LIN {X 0,Y 371.368,Z 260.473,A -85,B 0,C 180,E1 -13213.226,E2 -13213.226} C_VEL
LIN {X 0,Y 370.811,Z 274.455,A -85,B 0,C 180,E1 -13213.696,E2 -13213.696} C_VEL
LIN {X 0,Y 369.99,Z 288.054,A -85,B 0,C 180,E1 -13214.366,E2 -13214.366} C_VEL
LIN {X 0,Y 368.934,Z 301.272,A -85,B 0,C 180,E1 -13215.239,E2 -13215.239} C_VEL
LIN {X 0,Y 367.744,Z 313.996,A -85,B 0,C 180,E1 -13216.32,E2 -13216.32} C_VEL
LIN {X 0,Y 366.536,Z 325.561,A -85,B 0,C 180,E1 -13217.543,E2 -13217.543} C_VEL
LIN {X 0,Y 365.255,Z 336.172,A -85,B 0,C 180,E1 -13218.907,E2 -13218.907} C_VEL
LIN {X 0,Y 364.323,Z 345.06,A -85,B 0,C 180,E1 -13220.283,E2 -13220.283} C_VEL
LIN {X 0,Y 363.242,Z 354.016,A -85,B 0,C 180,E1 -13221.937,E2 -13221.937} C_VEL
LIN {X 0,Y 362.182,Z 362.593,A -85,B 0,C 180,E1 -13223.874,E2 -13223.874} C_VEL
LIN {X 0,Y 361.476,Z 368.625,A -85,B 0,C 180,E1 -13225.54,E2 -13225.54} C_VEL
LIN {X 0,Y 360.847,Z 375.044,A -85,B 0,C 180,E1 -13227.768,E2 -13227.768} C_VEL
LIN {X 0,Y 360.557,Z 379.848,A -85,B 0,C 180,E1 -13230,E2 -13230} C_VEL
LIN {X 0,Y 360.321,Z 383.186,A -85,B 0,C 180,E1 -13232.236,E2 -13232.236} C_VEL
LIN {X 0,Y 360.333,Z 385.14,A -85,B 0,C 180,E1 -13234.475,E2 -13234.475} C_VEL
LIN {X 0,Y 360.336,Z 385.758,A -85,B 0,C 180,E1 -13236.721,E2 -13236.721} C_VEL
LIN {X 0,Y 360.251,Z 385.048,A -85,B 0,C 180,E1 -13238.979,E2 -13238.979} C_VEL
LIN {X 0,Y 360.475,Z 382.984,A -85,B 0,C 180,E1 -13241.243,E2 -13241.243} C_VEL
LIN {X 0,Y 360.942,Z 379.51,A -85,B 0,C 180,E1 -13243.513,E2 -13243.513} C_VEL
LIN {X 0,Y 361.492,Z 374.512,A -85,B 0,C 180,E1 -13245.794,E2 -13245.794} C_VEL
LIN {X 0,Y 362.207,Z 369.647,A -85,B 0,C 180,E1 -13247.503,E2 -13247.503} C_VEL
LIN {X 0,Y 363.276,Z 362.599,A -85,B 0,C 180,E1 -13249.495,E2 -13249.495} C_VEL
LIN {X 0,Y 363.491,Z 361.022,A -85,B 0,C 180,E1 -13249.891,E2 -13249.891} C_VEL
LIN {X 0,Y 363.353,Z 357.833,A -85,B 0,C 180,E1 -13250.676,E2 -13250.676} C_VEL
LIN {X 0,Y 361.486,Z 352.461,A -85,B 0,C 180,E1 -13251.961,E2 -13251.961} C_VEL
LIN {X 0,Y 359.701,Z 346.613,A -85,B 0,C 180,E1 -13253.201,E2 -13253.201} C_VEL
LIN {X 0,Y 359.683,Z 342.682,A -85,B 0,C 180,E1 -13253.904,E2 -13253.904} C_VEL
LIN {X 0,Y 361.154,Z 332.979,A -85,B 0,C 180,E1 -13255.348,E2 -13255.348} C_VEL
LIN {X 0,Y 362.74,Z 322.514,A -85,B 0,C 180,E1 -13256.634,E2 -13256.634} C_VEL
LIN {X 0,Y 364.329,Z 309.965,A -85,B 0,C 180,E1 -13257.891,E2 -13257.891} C_VEL
LIN {X 0,Y 365.892,Z 297.682,A -85,B 0,C 180,E1 -13258.855,E2 -13258.855} C_VEL
LIN {X 0,Y 367.075,Z 284.046,A -85,B 0,C 180,E1 -13259.696,E2 -13259.696} C_VEL
LIN {X 0,Y 368.002,Z 270.326,A -85,B 0,C 180,E1 -13260.308,E2 -13260.308} C_VEL
LIN {X 0,Y 368.668,Z 256.311,A -85,B 0,C 180,E1 -13260.71,E2 -13260.71} C_VEL
LIN {X 0,Y 371.022,Z 157.916,A -85,B 0,C 180,E1 -13262.647,E2 -13262.647} C_VEL
LIN {X 0,Y 369.329,Z 151.129,A -85,B 0,C 180,E1 -13262.942,E2 -13262.942} C_VEL
LIN {X 0,Y 360.609,Z 131.607,A -85,B 0,C 180,E1 -13264.169,E2 -13264.169} C_VEL
LIN {X 0,Y 357.38,Z 124.729,A -85,B 0,C 180,E1 -13264.654,E2 -13264.654} C_VEL
LIN {X 0,Y 355.233,Z 116.033,A -85,B 0,C 180,E1 -13267.22,E2 -13267.22} C_VEL
LIN {X 0,Y 354.797,Z 114.414,A -85,B 0,C 180,E1 -13267.739,E2 -13267.739} C_VEL
LIN {X 0,Y 354.768,Z 114.419,A -85,B 0,C 180,E1 -13271.167,E2 -13271.167} C_VEL
LIN {X 0,Y 354.759,Z 114.419,A -85,B 0,C 180,E1 -13274.505,E2 -13274.505} C_VEL
LIN {X 0,Y 354.786,Z 114.42,A -85,B 0,C 180,E1 -13277.661,E2 -13277.661} C_VEL
LIN {X 0,Y 354.786,Z 114.4,A -85,B 0,C 180,E1 -13280.662,E2 -13280.662} C_VEL
LIN {X 0,Y 354.819,Z 114.407,A -85,B 0,C 180,E1 -13284.302,E2 -13284.302} C_VEL
LIN {X 0,Y 354.788,Z 114.416,A -85,B 0,C 180,E1 -13287.666,E2 -13287.666} C_VEL
LIN {X 0,Y 354.801,Z 114.414,A -85,B 0,C 180,E1 -13291.614,E2 -13291.614} C_VEL
LIN {X 0,Y 354.835,Z 114.409,A -85,B 0,C 180,E1 -13295.657,E2 -13295.657} C_VEL
LIN {X 0,Y 354.828,Z 114.412,A -85,B 0,C 180,E1 -13299.113,E2 -13299.113} C_VEL
LIN {X 0,Y 354.881,Z 114.4,A -85,B 0,C 180,E1 -13302.719,E2 -13302.719} C_VEL
LIN {X 0,Y 354.953,Z 114.388,A -85,B 0,C 180,E1 -13306.255,E2 -13306.255} C_VEL
LIN {X 0,Y 354.977,Z 114.392,A -85,B 0,C 180,E1 -13309.736,E2 -13309.736} C_VEL
LIN {X 0,Y 355.103,Z 114.375,A -85,B 0,C 180,E1 -13313.18,E2 -13313.18} C_VEL
LIN {X 0,Y 355.242,Z 114.356,A -85,B 0,C 180,E1 -13317.732,E2 -13317.732} C_VEL
LIN {X 0,Y 355.374,Z 114.338,A -85,B 0,C 180,E1 -13320,E2 -13320} C_VEL
LIN {X 0,Y 355.241,Z 114.355,A -85,B 0,C 180,E1 -13322.267,E2 -13322.267} C_VEL
LIN {X 0,Y 355.09,Z 114.368,A -85,B 0,C 180,E1 -13326.82,E2 -13326.82} C_VEL
LIN {X 0,Y 354.957,Z 114.389,A -85,B 0,C 180,E1 -13330.265,E2 -13330.265} C_VEL
LIN {X 0,Y 354.944,Z 114.395,A -85,B 0,C 180,E1 -13334.019,E2 -13334.019} C_VEL
LIN {X 0,Y 354.923,Z 114.396,A -85,B 0,C 180,E1 -13338.108,E2 -13338.108} C_VEL
LIN {X 0,Y 354.835,Z 114.405,A -85,B 0,C 180,E1 -13342.106,E2 -13342.106} C_VEL
LIN {X 0,Y 354.9,Z 114.397,A -85,B 0,C 180,E1 -13345.827,E2 -13345.827} C_VEL
LIN {X 0,Y 354.854,Z 114.404,A -85,B 0,C 180,E1 -13349.678,E2 -13349.678} C_VEL
LIN {X 0,Y 354.806,Z 114.412,A -85,B 0,C 180,E1 -13353.702,E2 -13353.702} C_VEL
LIN {X 0,Y 354.798,Z 114.413,A -85,B 0,C 180,E1 -13356.459,E2 -13356.459} C_VEL
LIN {X 0,Y 354.824,Z 114.393,A -85,B 0,C 180,E1 -13359.423,E2 -13359.423} C_VEL
LIN {X 0,Y 354.788,Z 114.414,A -85,B 0,C 180,E1 -13362.867,E2 -13362.867} C_VEL
LIN {X 0,Y 354.768,Z 114.417,A -85,B 0,C 180,E1 -13366.104,E2 -13366.104} C_VEL
LIN {X 0,Y 354.789,Z 114.414,A -85,B 0,C 180,E1 -13369.179,E2 -13369.179} C_VEL
LIN {X 0,Y 354.808,Z 114.409,A -85,B 0,C 180,E1 -13372.402,E2 -13372.402} C_VEL
LIN {X 0,Y 354.846,Z 114.473,A -85,B 0,C 180,E1 -13375.237,E2 -13375.237} C_VEL
LIN {X 0,Y 358.014,Z 126.781,A -85,B 0,C 180,E1 -13378.654,E2 -13378.654} C_VEL
LIN {X 0,Y 360.804,Z 138.768,A -85,B 0,C 180,E1 -13381.74,E2 -13381.74} C_VEL
LIN {X 0,Y 364.433,Z 147.556,A -85,B 0,C 180,E1 -13382.271,E2 -13382.271} C_VEL
LIN {X 0,Y 369.54,Z 172.482,A -85,B 0,C 180,E1 -13383.27,E2 -13383.27} C_VEL
LIN {X 0,Y 370.584,Z 178.889,A -85,B 0,C 180,E1 -13383.498,E2 -13383.498} C_VEL
LIN {X 0,Y 368.22,Z 276.377,A -85,B 0,C 180,E1 -13385.435,E2 -13385.435} C_VEL
LIN {X 0,Y 367.273,Z 291.024,A -85,B 0,C 180,E1 -13385.931,E2 -13385.931} C_VEL
LIN {X 0,Y 366.048,Z 304.419,A -85,B 0,C 180,E1 -13386.597,E2 -13386.597} C_VEL
LIN {X 0,Y 364.704,Z 317.241,A -85,B 0,C 180,E1 -13387.458,E2 -13387.458} C_VEL
LIN {X 0,Y 363.113,Z 330.167,A -85,B 0,C 180,E1 -13388.572,E2 -13388.572} C_VEL
LIN {X 0,Y 361.439,Z 341.712,A -85,B 0,C 180,E1 -13389.81,E2 -13389.81} C_VEL
LIN {X 0,Y 359.817,Z 352.311,A -85,B 0,C 180,E1 -13391.199,E2 -13391.199} C_VEL
LIN {X 0,Y 358.132,Z 362.837,A -85,B 0,C 180,E1 -13392.881,E2 -13392.881} C_VEL
LIN {X 0,Y 356.745,Z 371.541,A -85,B 0,C 180,E1 -13394.576,E2 -13394.576} C_VEL
LIN {X 0,Y 355.541,Z 379.91,A -85,B 0,C 180,E1 -13396.569,E2 -13396.569} C_VEL
LIN {X 0,Y 354.459,Z 386.661,A -85,B 0,C 180,E1 -13398.564,E2 -13398.564} C_VEL
LIN {X 0,Y 353.928,Z 391.311,A -85,B 0,C 180,E1 -13400.283,E2 -13400.283} C_VEL
LIN {X 0,Y 353.451,Z 396.148,A -85,B 0,C 180,E1 -13402.574,E2 -13402.574} C_VEL
LIN {X 0,Y 353.281,Z 398.78,A -85,B 0,C 180,E1 -13404.291,E2 -13404.291} C_VEL
LIN {X 0,Y 353.191,Z 401.09,A -85,B 0,C 180,E1 -13406.577,E2 -13406.577} C_VEL
LIN {X 0,Y 353.171,Z 402.06,A -85,B 0,C 180,E1 -13408.86,E2 -13408.86} C_VEL
LIN {X 0,Y 353.188,Z 401.7,A -85,B 0,C 180,E1 -13411.14,E2 -13411.14} C_VEL
LIN {X 0,Y 353.202,Z 399.998,A -85,B 0,C 180,E1 -13413.422,E2 -13413.422} C_VEL
LIN {X 0,Y 353.241,Z 396.911,A -85,B 0,C 180,E1 -13415.709,E2 -13415.709} C_VEL
LIN {X 0,Y 353.48,Z 392.343,A -85,B 0,C 180,E1 -13418,E2 -13418} C_VEL
LIN {X 0,Y 353.8,Z 387.808,A -85,B 0,C 180,E1 -13419.721,E2 -13419.721} C_VEL
LIN {X 0,Y 354.434,Z 381.27,A -85,B 0,C 180,E1 -13421.727,E2 -13421.727} C_VEL
LIN {X 0,Y 355.3,Z 373.143,A -85,B 0,C 180,E1 -13423.731,E2 -13423.731} C_VEL
LIN {X 0,Y 356.161,Z 364.616,A -85,B 0,C 180,E1 -13425.449,E2 -13425.449} C_VEL
LIN {X 0,Y 357.437,Z 354.324,A -85,B 0,C 180,E1 -13427.153,E2 -13427.153} C_VEL
LIN {X 0,Y 358.765,Z 343.962,A -85,B 0,C 180,E1 -13428.562,E2 -13428.562} C_VEL
LIN {X 0,Y 360.083,Z 332.707,A -85,B 0,C 180,E1 -13429.823,E2 -13429.823} C_VEL
LIN {X 0,Y 361.257,Z 320.946,A -85,B 0,C 180,E1 -13430.9,E2 -13430.9} C_VEL
LIN {X 0,Y 362.433,Z 307.882,A -85,B 0,C 180,E1 -13431.843,E2 -13431.843} C_VEL
LIN {X 0,Y 363.526,Z 293.919,A -85,B 0,C 180,E1 -13432.596,E2 -13432.596} C_VEL
LIN {X 0,Y 364.334,Z 279.288,A -85,B 0,C 180,E1 -13433.143,E2 -13433.143} C_VEL
LIN {X 0,Y 364.946,Z 256.943,A -85,B 0,C 180,E1 -13433.628,E2 -13433.628} C_VEL
LIN {X 0,Y 366.399,Z 176.054,A -85,B 0,C 180,E1 -13435.216,E2 -13435.216} C_VEL
LIN {X 0,Y 360.271,Z 140.609,A -85,B 0,C 180,E1 -13436.38,E2 -13436.38} C_VEL
LIN {X 0,Y 359.94,Z 138.758,A -85,B 0,C 180,E1 -13436.465,E2 -13436.465} C_VEL
LIN {X 0,Y 358.697,Z 131.582,A -85,B 0,C 180,E1 -13438.153,E2 -13438.153} C_VEL
LIN {X 0,Y 355.623,Z 117.892,A -85,B 0,C 180,E1 -13441.529,E2 -13441.529} C_VEL
LIN {X 0,Y 354.818,Z 114.415,A -85,B 0,C 180,E1 -13442.456,E2 -13442.456} C_VEL
LIN {X 0,Y 354.821,Z 114.413,A -85,B 0,C 180,E1 -13445.699,E2 -13445.699} C_VEL
LIN {X 0,Y 354.823,Z 114.41,A -85,B 0,C 180,E1 -13449.423,E2 -13449.423} C_VEL
LIN {X 0,Y 354.79,Z 114.413,A -85,B 0,C 180,E1 -13452.868,E2 -13452.868} C_VEL
LIN {X 0,Y 354.851,Z 114.407,A -85,B 0,C 180,E1 -13456.117,E2 -13456.117} C_VEL
LIN {X 0,Y 354.856,Z 114.406,A -85,B 0,C 180,E1 -13459.189,E2 -13459.189} C_VEL
LIN {X 0,Y 354.805,Z 114.41,A -85,B 0,C 180,E1 -13462.403,E2 -13462.403} C_VEL
LIN {X 0,Y 354.81,Z 114.411,A -85,B 0,C 180,E1 -13464.941,E2 -13464.941} C_VEL
LIN {X 0,Y 354.791,Z 114.412,A -85,B 0,C 180,E1 -13468.405,E2 -13468.405} C_VEL
LIN {X 0,Y 354.85,Z 114.408,A -85,B 0,C 180,E1 -13471.619,E2 -13471.619} C_VEL
LIN {X 0,Y 354.898,Z 114.399,A -85,B 0,C 180,E1 -13474.173,E2 -13474.173} C_VEL
LIN {X 0,Y 354.833,Z 114.407,A -85,B 0,C 180,E1 -13477.894,E2 -13477.894} C_VEL
LIN {X 0,Y 354.921,Z 114.395,A -85,B 0,C 180,E1 -13481.892,E2 -13481.892} C_VEL
LIN {X 0,Y 354.941,Z 114.394,A -85,B 0,C 180,E1 -13485.981,E2 -13485.981} C_VEL
LIN {X 0,Y 354.977,Z 114.389,A -85,B 0,C 180,E1 -13489.736,E2 -13489.736} C_VEL
LIN {X 0,Y 355.124,Z 114.371,A -85,B 0,C 180,E1 -13493.181,E2 -13493.181} C_VEL
LIN {X 0,Y 355.243,Z 114.357,A -85,B 0,C 180,E1 -13497.733,E2 -13497.733} C_VEL
LIN {X 0,Y 355.395,Z 114.34,A -85,B 0,C 180,E1 -13500,E2 -13500} C_VEL
LIN {X 0,Y 355.243,Z 114.36,A -85,B 0,C 180,E1 -13502.268,E2 -13502.268} C_VEL
LIN {X 0,Y 355.102,Z 114.374,A -85,B 0,C 180,E1 -13506.82,E2 -13506.82} C_VEL
LIN {X 0,Y 354.977,Z 114.391,A -85,B 0,C 180,E1 -13510.264,E2 -13510.264} C_VEL
LIN {X 0,Y 354.942,Z 114.398,A -85,B 0,C 180,E1 -13514.019,E2 -13514.019} C_VEL
LIN {X 0,Y 354.922,Z 114.397,A -85,B 0,C 180,E1 -13518.109,E2 -13518.109} C_VEL
LIN {X 0,Y 354.835,Z 114.408,A -85,B 0,C 180,E1 -13522.106,E2 -13522.106} C_VEL
LIN {X 0,Y 354.899,Z 114.401,A -85,B 0,C 180,E1 -13525.828,E2 -13525.828} C_VEL
LIN {X 0,Y 354.817,Z 114.411,A -85,B 0,C 180,E1 -13529.682,E2 -13529.682} C_VEL
LIN {X 0,Y 354.806,Z 114.412,A -85,B 0,C 180,E1 -13533.702,E2 -13533.702} C_VEL
LIN {X 0,Y 354.797,Z 114.412,A -85,B 0,C 180,E1 -13536.46,E2 -13536.46} C_VEL
LIN {X 0,Y 354.824,Z 114.411,A -85,B 0,C 180,E1 -13539.424,E2 -13539.424} C_VEL
LIN {X 0,Y 354.789,Z 114.418,A -85,B 0,C 180,E1 -13542.868,E2 -13542.868} C_VEL
LIN {X 0,Y 354.768,Z 114.415,A -85,B 0,C 180,E1 -13546.104,E2 -13546.104} C_VEL
LIN {X 0,Y 354.787,Z 114.414,A -85,B 0,C 180,E1 -13549.179,E2 -13549.179} C_VEL
LIN {X 0,Y 354.807,Z 114.413,A -85,B 0,C 180,E1 -13552.403,E2 -13552.403} C_VEL
LIN {X 0,Y 354.813,Z 114.412,A -85,B 0,C 180,E1 -13554.941,E2 -13554.941} C_VEL
LIN {X 0,Y 354.795,Z 114.418,A -85,B 0,C 180,E1 -13558.406,E2 -13558.406} C_VEL
LIN {X 0,Y 354.803,Z 114.412,A -85,B 0,C 180,E1 -13561.615,E2 -13561.615} C_VEL
LIN {X 0,Y 354.836,Z 114.409,A -85,B 0,C 180,E1 -13565.657,E2 -13565.657} C_VEL
LIN {X 0,Y 354.894,Z 114.59,A -85,B 0,C 180,E1 -13566.745,E2 -13566.745} C_VEL
LIN {X 0,Y 357.071,Z 124.538,A -85,B 0,C 180,E1 -13569.419,E2 -13569.419} C_VEL
LIN {X 0,Y 364.492,Z 143.98,A -85,B 0,C 180,E1 -13570.358,E2 -13570.358} C_VEL
LIN {X 0,Y 366.9,Z 156.799,A -85,B 0,C 180,E1 -13570.79,E2 -13570.79} C_VEL
LIN {X 0,Y 364.744,Z 260.78,A -85,B 0,C 180,E1 -13572.84,E2 -13572.84} C_VEL
LIN {X 0,Y 364.132,Z 275.452,A -85,B 0,C 180,E1 -13573.352,E2 -13573.352} C_VEL
LIN {X 0,Y 363.2,Z 289.405,A -85,B 0,C 180,E1 -13574.066,E2 -13574.066} C_VEL
LIN {X 0,Y 362.109,Z 302.365,A -85,B 0,C 180,E1 -13574.955,E2 -13574.955} C_VEL
LIN {X 0,Y 360.91,Z 314.908,A -85,B 0,C 180,E1 -13576.056,E2 -13576.056} C_VEL
LIN {X 0,Y 359.669,Z 326.341,A -85,B 0,C 180,E1 -13577.301,E2 -13577.301} C_VEL
LIN {X 0,Y 358.271,Z 337.358,A -85,B 0,C 180,E1 -13578.763,E2 -13578.763} C_VEL
LIN {X 0,Y 357.157,Z 347.266,A -85,B 0,C 180,E1 -13580.372,E2 -13580.372} C_VEL
LIN {X 0,Y 356.017,Z 355.883,A -85,B 0,C 180,E1 -13582.057,E2 -13582.057} C_VEL
LIN {X 0,Y 355.031,Z 364.157,A -85,B 0,C 180,E1 -13584.035,E2 -13584.035} C_VEL
LIN {X 0,Y 354.242,Z 370.815,A -85,B 0,C 180,E1 -13586.018,E2 -13586.018} C_VEL
LIN {X 0,Y 353.689,Z 376.731,A -85,B 0,C 180,E1 -13588.292,E2 -13588.292} C_VEL
LIN {X 0,Y 353.47,Z 380.152,A -85,B 0,C 180,E1 -13590,E2 -13590} C_VEL
LIN {X 0,Y 353.224,Z 383.442,A -85,B 0,C 180,E1 -13592.281,E2 -13592.281} C_VEL
LIN {X 0,Y 353.246,Z 385.341,A -85,B 0,C 180,E1 -13594.565,E2 -13594.565} C_VEL
LIN {X 0,Y 353.226,Z 385.912,A -85,B 0,C 180,E1 -13596.856,E2 -13596.856} C_VEL
LIN {X 0,Y 353.163,Z 385.158,A -85,B 0,C 180,E1 -13599.161,E2 -13599.161} C_VEL
LIN {X 0,Y 353.438,Z 383.051,A -85,B 0,C 180,E1 -13601.47,E2 -13601.47} C_VEL
LIN {X 0,Y 353.91,Z 379.531,A -85,B 0,C 180,E1 -13603.786,E2 -13603.786} C_VEL
LIN {X 0,Y 354.52,Z 374.484,A -85,B 0,C 180,E1 -13606.113,E2 -13606.113} C_VEL
LIN {X 0,Y 355.29,Z 369.566,A -85,B 0,C 180,E1 -13607.855,E2 -13607.855} C_VEL
LIN {X 0,Y 356.428,Z 362.461,A -85,B 0,C 180,E1 -13609.885,E2 -13609.885} C_VEL
LIN {X 0,Y 357.633,Z 354.998,A -85,B 0,C 180,E1 -13611.621,E2 -13611.621} C_VEL
LIN {X 0,Y 359.168,Z 345.993,A -85,B 0,C 180,E1 -13613.344,E2 -13613.344} C_VEL
LIN {X 0,Y 359.683,Z 342.682,A -85,B 0,C 180,E1 -13613.904,E2 -13613.904} C_VEL
LIN {X 0,Y 359.684,Z 338.612,A -85,B 0,C 180,E1 -13614.586,E2 -13614.586} C_VEL
LIN {X 0,Y 358.044,Z 331.879,A -85,B 0,C 180,E1 -13615.721,E2 -13615.721} C_VEL
LIN {X 0,Y 356.488,Z 324.785,A -85,B 0,C 180,E1 -13616.791,E2 -13616.791} C_VEL
LIN {X 0,Y 356.6,Z 320.066,A -85,B 0,C 180,E1 -13617.363,E2 -13617.363} C_VEL
LIN {X 0,Y 358.195,Z 307.689,A -85,B 0,C 180,E1 -13618.571,E2 -13618.571} C_VEL
LIN {X 0,Y 359.791,Z 294.774,A -85,B 0,C 180,E1 -13619.553,E2 -13619.553} C_VEL
LIN {X 0,Y 360.938,Z 281.508,A -85,B 0,C 180,E1 -13620.334,E2 -13620.334} C_VEL
LIN {X 0,Y 361.892,Z 267.219,A -85,B 0,C 180,E1 -13620.927,E2 -13620.927} C_VEL
LIN {X 0,Y 362.475,Z 252.016,A -85,B 0,C 180,E1 -13621.315,E2 -13621.315} C_VEL
LIN {X 0,Y 364.784,Z 158.967,A -85,B 0,C 180,E1 -13623.171,E2 -13623.171} C_VEL
LIN {X 0,Y 363.36,Z 153.69,A -85,B 0,C 180,E1 -13623.416,E2 -13623.416} C_VEL
LIN {X 0,Y 355.153,Z 135.268,A -85,B 0,C 180,E1 -13624.608,E2 -13624.608} C_VEL
LIN {X 0,Y 350.218,Z 124.881,A -85,B 0,C 180,E1 -13625.371,E2 -13625.371} C_VEL
LIN {X 0,Y 347.731,Z 115.296,A -85,B 0,C 180,E1 -13628.339,E2 -13628.339} C_VEL
LIN {X 0,Y 347.741,Z 115.295,A -85,B 0,C 180,E1 -13631.832,E2 -13631.832} C_VEL
LIN {X 0,Y 347.701,Z 115.291,A -85,B 0,C 180,E1 -13635.028,E2 -13635.028} C_VEL
LIN {X 0,Y 347.74,Z 115.293,A -85,B 0,C 180,E1 -13638.399,E2 -13638.399} C_VEL
LIN {X 0,Y 347.763,Z 115.291,A -85,B 0,C 180,E1 -13642.014,E2 -13642.014} C_VEL
LIN {X 0,Y 347.744,Z 115.294,A -85,B 0,C 180,E1 -13645.536,E2 -13645.536} C_VEL
LIN {X 0,Y 347.746,Z 115.292,A -85,B 0,C 180,E1 -13648.3,E2 -13648.3} C_VEL
LIN {X 0,Y 347.747,Z 115.29,A -85,B 0,C 180,E1 -13650.984,E2 -13650.984} C_VEL
LIN {X 0,Y 347.749,Z 115.285,A -85,B 0,C 180,E1 -13653.601,E2 -13653.601} C_VEL
LIN {X 0,Y 347.764,Z 115.291,A -85,B 0,C 180,E1 -13656.16,E2 -13656.16} C_VEL
LIN {X 0,Y 347.807,Z 115.285,A -85,B 0,C 180,E1 -13659.909,E2 -13659.909} C_VEL
LIN {X 0,Y 347.833,Z 115.281,A -85,B 0,C 180,E1 -13663.568,E2 -13663.568} C_VEL
LIN {X 0,Y 347.891,Z 115.271,A -85,B 0,C 180,E1 -13667.16,E2 -13667.16} C_VEL
LIN {X 0,Y 347.941,Z 115.258,A -85,B 0,C 180,E1 -13670.701,E2 -13670.701} C_VEL
LIN {X 0,Y 348.053,Z 115.255,A -85,B 0,C 180,E1 -13674.205,E2 -13674.205} C_VEL
LIN {X 0,Y 348.204,Z 115.232,A -85,B 0,C 180,E1 -13677.686,E2 -13677.686} C_VEL
LIN {X 0,Y 348.324,Z 115.216,A -85,B 0,C 180,E1 -13680,E2 -13680} C_VEL
LIN {X 0,Y 348.203,Z 115.232,A -85,B 0,C 180,E1 -13682.313,E2 -13682.313} C_VEL
LIN {X 0,Y 348.056,Z 115.244,A -85,B 0,C 180,E1 -13686.958,E2 -13686.958} C_VEL
LIN {X 0,Y 347.897,Z 115.268,A -85,B 0,C 180,E1 -13690.475,E2 -13690.475} C_VEL
LIN {X 0,Y 347.899,Z 115.272,A -85,B 0,C 180,E1 -13694.15,E2 -13694.15} C_VEL
LIN {X 0,Y 347.891,Z 115.272,A -85,B 0,C 180,E1 -13698.29,E2 -13698.29} C_VEL
LIN {X 0,Y 347.79,Z 115.282,A -85,B 0,C 180,E1 -13701.635,E2 -13701.635} C_VEL
LIN {X 0,Y 347.813,Z 115.276,A -85,B 0,C 180,E1 -13705.108,E2 -13705.108} C_VEL
LIN {X 0,Y 347.811,Z 115.281,A -85,B 0,C 180,E1 -13707.694,E2 -13707.694} C_VEL
LIN {X 0,Y 347.764,Z 115.289,A -85,B 0,C 180,E1 -13710.346,E2 -13710.346} C_VEL
LIN {X 0,Y 347.745,Z 115.295,A -85,B 0,C 180,E1 -13714.464,E2 -13714.464} C_VEL
LIN {X 0,Y 347.773,Z 115.288,A -85,B 0,C 180,E1 -13717.988,E2 -13717.988} C_VEL
LIN {X 0,Y 347.751,Z 115.291,A -85,B 0,C 180,E1 -13721.83,E2 -13721.83} C_VEL
LIN {X 0,Y 347.706,Z 115.286,A -85,B 0,C 180,E1 -13725.027,E2 -13725.027} C_VEL
LIN {X 0,Y 347.751,Z 115.295,A -85,B 0,C 180,E1 -13728.397,E2 -13728.397} C_VEL
LIN {X 0,Y 347.774,Z 115.287,A -85,B 0,C 180,E1 -13732.011,E2 -13732.011} C_VEL
LIN {X 0,Y 347.814,Z 115.462,A -85,B 0,C 180,E1 -13734.662,E2 -13734.662} C_VEL
LIN {X 0,Y 350.854,Z 127.145,A -85,B 0,C 180,E1 -13738.005,E2 -13738.005} C_VEL
LIN {X 0,Y 353.561,Z 138.61,A -85,B 0,C 180,E1 -13741.042,E2 -13741.042} C_VEL
LIN {X 0,Y 358.571,Z 150.353,A -85,B 0,C 180,E1 -13741.794,E2 -13741.794} C_VEL
LIN {X 0,Y 363.378,Z 173.831,A -85,B 0,C 180,E1 -13742.762,E2 -13742.762} C_VEL
LIN {X 0,Y 364.349,Z 179.267,A -85,B 0,C 180,E1 -13742.969,E2 -13742.969} C_VEL
LIN {X 0,Y 361.877,Z 276.592,A -85,B 0,C 180,E1 -13744.937,E2 -13744.937} C_VEL
LIN {X 0,Y 360.891,Z 291.105,A -85,B 0,C 180,E1 -13745.44,E2 -13745.44} C_VEL
LIN {X 0,Y 359.585,Z 304.996,A -85,B 0,C 180,E1 -13746.151,E2 -13746.151} C_VEL
LIN {X 0,Y 358.154,Z 317.742,A -85,B 0,C 180,E1 -13747.029,E2 -13747.029} C_VEL
LIN {X 0,Y 356.525,Z 330.47,A -85,B 0,C 180,E1 -13748.156,E2 -13748.156} C_VEL
LIN {X 0,Y 354.789,Z 341.932,A -85,B 0,C 180,E1 -13749.414,E2 -13749.414} C_VEL
LIN {X 0,Y 353.101,Z 352.464,A -85,B 0,C 180,E1 -13750.828,E2 -13750.828} C_VEL
LIN {X 0,Y 351.319,Z 362.937,A -85,B 0,C 180,E1 -13752.538,E2 -13752.538} C_VEL
LIN {X 0,Y 349.856,Z 371.597,A -85,B 0,C 180,E1 -13754.265,E2 -13754.265} C_VEL
LIN {X 0,Y 348.585,Z 379.925,A -85,B 0,C 180,E1 -13756.296,E2 -13756.296} C_VEL
LIN {X 0,Y 347.468,Z 386.637,A -85,B 0,C 180,E1 -13758.331,E2 -13758.331} C_VEL
LIN {X 0,Y 346.736,Z 392.612,A -85,B 0,C 180,E1 -13760.668,E2 -13760.668} C_VEL
LIN {X 0,Y 346.319,Z 397.016,A -85,B 0,C 180,E1 -13763.006,E2 -13763.006} C_VEL
LIN {X 0,Y 346.138,Z 399.986,A -85,B 0,C 180,E1 -13765.341,E2 -13765.341} C_VEL
LIN {X 0,Y 346.066,Z 401.597,A -85,B 0,C 180,E1 -13767.672,E2 -13767.672} C_VEL
LIN {X 0,Y 346.113,Z 401.878,A -85,B 0,C 180,E1 -13770,E2 -13770} C_VEL
LIN {X 0,Y 346.076,Z 400.823,A -85,B 0,C 180,E1 -13772.328,E2 -13772.328} C_VEL
LIN {X 0,Y 346.128,Z 398.412,A -85,B 0,C 180,E1 -13774.658,E2 -13774.658} C_VEL
LIN {X 0,Y 346.261,Z 394.572,A -85,B 0,C 180,E1 -13776.995,E2 -13776.995} C_VEL
LIN {X 0,Y 346.513,Z 390.635,A -85,B 0,C 180,E1 -13778.749,E2 -13778.749} C_VEL
LIN {X 0,Y 347.073,Z 383.955,A -85,B 0,C 180,E1 -13781.091,E2 -13781.091} C_VEL
LIN {X 0,Y 347.88,Z 376.504,A -85,B 0,C 180,E1 -13783.137,E2 -13783.137} C_VEL
LIN {X 0,Y 348.707,Z 368.798,A -85,B 0,C 180,E1 -13784.866,E2 -13784.866} C_VEL
LIN {X 0,Y 349.944,Z 359.292,A -85,B 0,C 180,E1 -13786.63,E2 -13786.63} C_VEL
LIN {X 0,Y 351.138,Z 348.863,A -85,B 0,C 180,E1 -13788.224,E2 -13788.224} C_VEL
LIN {X 0,Y 352.534,Z 338.664,A -85,B 0,C 180,E1 -13789.507,E2 -13789.507} C_VEL
LIN {X 0,Y 353.955,Z 326.221,A -85,B 0,C 180,E1 -13790.788,E2 -13790.788} C_VEL
LIN {X 0,Y 355.228,Z 314.085,A -85,B 0,C 180,E1 -13791.786,E2 -13791.786} C_VEL
LIN {X 0,Y 356.298,Z 301.099,A -85,B 0,C 180,E1 -13792.621,E2 -13792.621} C_VEL
LIN {X 0,Y 357.289,Z 286.955,A -85,B 0,C 180,E1 -13793.281,E2 -13793.281} C_VEL
LIN {X 0,Y 357.991,Z 272.032,A -85,B 0,C 180,E1 -13793.731,E2 -13793.731} C_VEL
LIN {X 0,Y 359.918,Z 177.39,A -85,B 0,C 180,E1 -13795.62,E2 -13795.62} C_VEL
LIN {X 0,Y 354.009,Z 142.834,A -85,B 0,C 180,E1 -13796.781,E2 -13796.781} C_VEL
LIN {X 0,Y 352.889,Z 138.564,A -85,B 0,C 180,E1 -13796.984,E2 -13796.984} C_VEL
LIN {X 0,Y 350.207,Z 125.859,A -85,B 0,C 180,E1 -13800.112,E2 -13800.112} C_VEL
LIN {X 0,Y 347.779,Z 115.29,A -85,B 0,C 180,E1 -13802.855,E2 -13802.855} C_VEL
LIN {X 0,Y 347.77,Z 115.294,A -85,B 0,C 180,E1 -13806.065,E2 -13806.065} C_VEL
LIN {X 0,Y 347.751,Z 115.291,A -85,B 0,C 180,E1 -13808.792,E2 -13808.792} C_VEL
LIN {X 0,Y 347.75,Z 115.295,A -85,B 0,C 180,E1 -13811.83,E2 -13811.83} C_VEL
LIN {X 0,Y 347.796,Z 115.284,A -85,B 0,C 180,E1 -13815.011,E2 -13815.011} C_VEL
LIN {X 0,Y 347.785,Z 115.286,A -85,B 0,C 180,E1 -13818.39,E2 -13818.39} C_VEL
LIN {X 0,Y 347.772,Z 115.287,A -85,B 0,C 180,E1 -13822.011,E2 -13822.011} C_VEL
LIN {X 0,Y 347.743,Z 115.295,A -85,B 0,C 180,E1 -13825.536,E2 -13825.536} C_VEL
LIN {X 0,Y 347.762,Z 115.29,A -85,B 0,C 180,E1 -13829.654,E2 -13829.654} C_VEL
LIN {X 0,Y 347.85,Z 115.279,A -85,B 0,C 180,E1 -13832.745,E2 -13832.745} C_VEL
LIN {X 0,Y 347.787,Z 115.284,A -85,B 0,C 180,E1 -13836.162,E2 -13836.162} C_VEL
LIN {X 0,Y 347.811,Z 115.282,A -85,B 0,C 180,E1 -13839.909,E2 -13839.909} C_VEL
LIN {X 0,Y 347.865,Z 115.275,A -85,B 0,C 180,E1 -13842.359,E2 -13842.359} C_VEL
LIN {X 0,Y 347.896,Z 115.271,A -85,B 0,C 180,E1 -13845.971,E2 -13845.971} C_VEL
LIN {X 0,Y 347.927,Z 115.267,A -85,B 0,C 180,E1 -13849.526,E2 -13849.526} C_VEL
LIN {X 0,Y 348.09,Z 115.247,A -85,B 0,C 180,E1 -13853.042,E2 -13853.042} C_VEL
LIN {X 0,Y 348.205,Z 115.234,A -85,B 0,C 180,E1 -13857.687,E2 -13857.687} C_VEL
LIN {X 0,Y 348.344,Z 115.218,A -85,B 0,C 180,E1 -13860,E2 -13860} C_VEL
LIN {X 0,Y 348.205,Z 115.236,A -85,B 0,C 180,E1 -13862.314,E2 -13862.314} C_VEL
LIN {X 0,Y 348.069,Z 115.25,A -85,B 0,C 180,E1 -13866.959,E2 -13866.959} C_VEL
LIN {X 0,Y 347.928,Z 115.267,A -85,B 0,C 180,E1 -13870.475,E2 -13870.475} C_VEL
LIN {X 0,Y 347.898,Z 115.274,A -85,B 0,C 180,E1 -13874.15,E2 -13874.15} C_VEL
LIN {X 0,Y 347.89,Z 115.272,A -85,B 0,C 180,E1 -13878.29,E2 -13878.29} C_VEL
LIN {X 0,Y 347.79,Z 115.29,A -85,B 0,C 180,E1 -13881.636,E2 -13881.636} C_VEL
LIN {X 0,Y 347.812,Z 115.283,A -85,B 0,C 180,E1 -13885.109,E2 -13885.109} C_VEL
LIN {X 0,Y 347.808,Z 115.286,A -85,B 0,C 180,E1 -13887.694,E2 -13887.694} C_VEL
LIN {X 0,Y 347.749,Z 115.289,A -85,B 0,C 180,E1 -13890.348,E2 -13890.348} C_VEL
LIN {X 0,Y 347.748,Z 115.29,A -85,B 0,C 180,E1 -13894.044,E2 -13894.044} C_VEL
LIN {X 0,Y 347.761,Z 115.291,A -85,B 0,C 180,E1 -13897.321,E2 -13897.321} C_VEL
LIN {X 0,Y 347.732,Z 115.293,A -85,B 0,C 180,E1 -13900.297,E2 -13900.297} C_VEL
LIN {X 0,Y 347.727,Z 115.294,A -85,B 0,C 180,E1 -13903.408,E2 -13903.408} C_VEL
LIN {X 0,Y 347.726,Z 115.297,A -85,B 0,C 180,E1 -13906.687,E2 -13906.687} C_VEL
LIN {X 0,Y 347.747,Z 115.291,A -85,B 0,C 180,E1 -13910.174,E2 -13910.174} C_VEL
LIN {X 0,Y 347.761,Z 115.293,A -85,B 0,C 180,E1 -13912.68,E2 -13912.68} C_VEL
LIN {X 0,Y 347.749,Z 115.291,A -85,B 0,C 180,E1 -13915.957,E2 -13915.957} C_VEL
LIN {X 0,Y 347.742,Z 115.292,A -85,B 0,C 180,E1 -13919.652,E2 -13919.652} C_VEL
LIN {X 0,Y 347.752,Z 115.29,A -85,B 0,C 180,E1 -13923.602,E2 -13923.602} C_VEL
LIN {X 0,Y 347.843,Z 115.401,A -85,B 0,C 180,E1 -13926.324,E2 -13926.324} C_VEL
LIN {X 0,Y 349.958,Z 124.852,A -85,B 0,C 180,E1 -13928.896,E2 -13928.896} C_VEL
LIN {X 0,Y 357.973,Z 145.511,A -85,B 0,C 180,E1 -13929.936,E2 -13929.936} C_VEL
LIN {X 0,Y 360.385,Z 157.192,A -85,B 0,C 180,E1 -13930.356,E2 -13930.356} C_VEL
LIN {X 0,Y 358.115,Z 261.076,A -85,B 0,C 180,E1 -13932.438,E2 -13932.438} C_VEL
LIN {X 0,Y 357.504,Z 275.688,A -85,B 0,C 180,E1 -13932.96,E2 -13932.96} C_VEL
LIN {X 0,Y 356.536,Z 289.624,A -85,B 0,C 180,E1 -13933.687,E2 -13933.687} C_VEL
LIN {X 0,Y 355.306,Z 303.452,A -85,B 0,C 180,E1 -13934.659,E2 -13934.659} C_VEL
LIN {X 0,Y 354.087,Z 315.814,A -85,B 0,C 180,E1 -13935.782,E2 -13935.782} C_VEL
LIN {X 0,Y 352.656,Z 328.28,A -85,B 0,C 180,E1 -13937.191,E2 -13937.191} C_VEL
LIN {X 0,Y 351.352,Z 338.184,A -85,B 0,C 180,E1 -13938.562,E2 -13938.562} C_VEL
LIN {X 0,Y 350.193,Z 347.856,A -85,B 0,C 180,E1 -13940.178,E2 -13940.178} C_VEL
LIN {X 0,Y 349.01,Z 356.403,A -85,B 0,C 180,E1 -13941.897,E2 -13941.897} C_VEL
LIN {X 0,Y 348.013,Z 364.601,A -85,B 0,C 180,E1 -13943.914,E2 -13943.914} C_VEL
LIN {X 0,Y 347.19,Z 371.198,A -85,B 0,C 180,E1 -13945.937,E2 -13945.937} C_VEL
LIN {X 0,Y 346.617,Z 377.058,A -85,B 0,C 180,E1 -13948.257,E2 -13948.257} C_VEL
LIN {X 0,Y 346.385,Z 380.456,A -85,B 0,C 180,E1 -13950,E2 -13950} C_VEL
LIN {X 0,Y 346.131,Z 383.688,A -85,B 0,C 180,E1 -13952.328,E2 -13952.328} C_VEL
LIN {X 0,Y 346.144,Z 385.536,A -85,B 0,C 180,E1 -13954.659,E2 -13954.659} C_VEL
LIN {X 0,Y 346.199,Z 385.972,A -85,B 0,C 180,E1 -13955.885,E2 -13955.885} C_VEL
LIN {X 0,Y 346.087,Z 385.834,A -85,B 0,C 180,E1 -13958.172,E2 -13958.172} C_VEL
LIN {X 0,Y 346.163,Z 384.365,A -85,B 0,C 180,E1 -13960.529,E2 -13960.529} C_VEL
LIN {X 0,Y 346.642,Z 381.518,A -85,B 0,C 180,E1 -13962.887,E2 -13962.887} C_VEL
LIN {X 0,Y 347.172,Z 377.206,A -85,B 0,C 180,E1 -13965.258,E2 -13965.258} C_VEL
LIN {X 0,Y 348.123,Z 371.286,A -85,B 0,C 180,E1 -13967.627,E2 -13967.627} C_VEL
LIN {X 0,Y 349.249,Z 364.573,A -85,B 0,C 180,E1 -13969.698,E2 -13969.698} C_VEL
LIN {X 0,Y 350.663,Z 356.166,A -85,B 0,C 180,E1 -13971.764,E2 -13971.764} C_VEL
LIN {X 0,Y 352.234,Z 347.367,A -85,B 0,C 180,E1 -13973.519,E2 -13973.519} C_VEL
LIN {X 0,Y 353.946,Z 336.656,A -85,B 0,C 180,E1 -13975.272,E2 -13975.272} C_VEL
LIN {X 0,Y 355.694,Z 325.806,A -85,B 0,C 180,E1 -13976.712,E2 -13976.712} C_VEL
LIN {X 0,Y 356.6,Z 320.066,A -85,B 0,C 180,E1 -13977.363,E2 -13977.363} C_VEL
LIN {X 0,Y 356.443,Z 316.886,A -85,B 0,C 180,E1 -13977.75,E2 -13977.75} C_VEL
LIN {X 0,Y 352.515,Z 306.935,A -85,B 0,C 180,E1 -13979.092,E2 -13979.092} C_VEL
LIN {X 0,Y 352.36,Z 303.512,A -85,B 0,C 180,E1 -13979.419,E2 -13979.419} C_VEL
LIN {X 0,Y 353.796,Z 290.433,A -85,B 0,C 180,E1 -13980.352,E2 -13980.352} C_VEL
LIN {X 0,Y 354.997,Z 276.305,A -85,B 0,C 180,E1 -13981.102,E2 -13981.102} C_VEL
LIN {X 0,Y 355.889,Z 261.563,A -85,B 0,C 180,E1 -13981.63,E2 -13981.63} C_VEL
LIN {X 0,Y 358.698,Z 160.682,A -85,B 0,C 180,E1 -13983.687,E2 -13983.687} C_VEL
LIN {X 0,Y 357.493,Z 156.399,A -85,B 0,C 180,E1 -13983.897,E2 -13983.897} C_VEL
LIN {X 0,Y 349.512,Z 138.471,A -85,B 0,C 180,E1 -13985.092,E2 -13985.092} C_VEL
LIN {X 0,Y 343.035,Z 125.173,A -85,B 0,C 180,E1 -13986.09,E2 -13986.09} C_VEL
LIN {X 0,Y 340.694,Z 116.172,A -85,B 0,C 180,E1 -13988.968,E2 -13988.968} C_VEL
LIN {X 0,Y 340.673,Z 116.174,A -85,B 0,C 180,E1 -13992.905,E2 -13992.905} C_VEL
LIN {X 0,Y 340.673,Z 116.171,A -85,B 0,C 180,E1 -13997.095,E2 -13997.095} C_VEL
LIN {X 0,Y 340.656,Z 116.158,A -85,B 0,C 180,E1 -14000.241,E2 -14000.241} C_VEL
LIN {X 0,Y 340.708,Z 116.167,A -85,B 0,C 180,E1 -14003.56,E2 -14003.56} C_VEL
LIN {X 0,Y 340.693,Z 116.17,A -85,B 0,C 180,E1 -14006.153,E2 -14006.153} C_VEL
LIN {X 0,Y 340.725,Z 116.161,A -85,B 0,C 180,E1 -14010.034,E2 -14010.034} C_VEL
LIN {X 0,Y 340.72,Z 116.164,A -85,B 0,C 180,E1 -14013.012,E2 -14013.012} C_VEL
LIN {X 0,Y 340.74,Z 116.165,A -85,B 0,C 180,E1 -14015.637,E2 -14015.637} C_VEL
LIN {X 0,Y 340.735,Z 116.166,A -85,B 0,C 180,E1 -14019.473,E2 -14019.473} C_VEL
LIN {X 0,Y 340.794,Z 116.149,A -85,B 0,C 180,E1 -14021.98,E2 -14021.98} C_VEL
LIN {X 0,Y 340.871,Z 116.144,A -85,B 0,C 180,E1 -14025.705,E2 -14025.705} C_VEL
LIN {X 0,Y 340.871,Z 116.148,A -85,B 0,C 180,E1 -14029.306,E2 -14029.306} C_VEL
LIN {X 0,Y 341.012,Z 116.131,A -85,B 0,C 180,E1 -14032.897,E2 -14032.897} C_VEL
LIN {X 0,Y 340.834,Z 116.149,A -85,B 0,C 180,E1 -14035.269,E2 -14035.269} C_VEL
LIN {X 0,Y 341.165,Z 116.108,A -85,B 0,C 180,E1 -14037.639,E2 -14037.639} C_VEL
LIN {X 0,Y 341.275,Z 116.094,A -85,B 0,C 180,E1 -14040,E2 -14040} C_VEL
LIN {X 0,Y 341.165,Z 116.109,A -85,B 0,C 180,E1 -14042.361,E2 -14042.361} C_VEL
LIN {X 0,Y 341.003,Z 116.123,A -85,B 0,C 180,E1 -14047.103,E2 -14047.103} C_VEL
LIN {X 0,Y 340.849,Z 116.146,A -85,B 0,C 180,E1 -14050.694,E2 -14050.694} C_VEL
LIN {X 0,Y 340.864,Z 116.148,A -85,B 0,C 180,E1 -14054.325,E2 -14054.325} C_VEL
LIN {X 0,Y 340.838,Z 116.151,A -85,B 0,C 180,E1 -14058.466,E2 -14058.466} C_VEL
LIN {X 0,Y 340.754,Z 116.16,A -85,B 0,C 180,E1 -14061.857,E2 -14061.857} C_VEL
LIN {X 0,Y 340.773,Z 116.156,A -85,B 0,C 180,E1 -14065.664,E2 -14065.664} C_VEL
LIN {X 0,Y 340.742,Z 116.16,A -85,B 0,C 180,E1 -14068.319,E2 -14068.319} C_VEL
LIN {X 0,Y 340.704,Z 116.169,A -85,B 0,C 180,E1 -14071.044,E2 -14071.044} C_VEL
LIN {X 0,Y 340.718,Z 116.163,A -85,B 0,C 180,E1 -14075.279,E2 -14075.279} C_VEL
LIN {X 0,Y 340.709,Z 116.16,A -85,B 0,C 180,E1 -14078.386,E2 -14078.386} C_VEL
LIN {X 0,Y 340.699,Z 116.171,A -85,B 0,C 180,E1 -14082.045,E2 -14082.045} C_VEL
LIN {X 0,Y 340.652,Z 116.176,A -85,B 0,C 180,E1 -14086.227,E2 -14086.227} C_VEL
LIN {X 0,Y 340.689,Z 116.171,A -85,B 0,C 180,E1 -14089.753,E2 -14089.753} C_VEL
LIN {X 0,Y 340.706,Z 116.167,A -85,B 0,C 180,E1 -14093.258,E2 -14093.258} C_VEL
LIN {X 0,Y 340.771,Z 116.257,A -85,B 0,C 180,E1 -14094,E2 -14094} C_VEL
LIN {X 0,Y 343.421,Z 126.529,A -85,B 0,C 180,E1 -14097.04,E2 -14097.04} C_VEL
LIN {X 0,Y 346.172,Z 137.811,A -85,B 0,C 180,E1 -14100.189,E2 -14100.189} C_VEL
LIN {X 0,Y 346.393,Z 138.621,A -85,B 0,C 180,E1 -14100.321,E2 -14100.321} C_VEL
LIN {X 0,Y 352.712,Z 152.863,A -85,B 0,C 180,E1 -14101.291,E2 -14101.291} C_VEL
LIN {X 0,Y 357.62,Z 177.455,A -85,B 0,C 180,E1 -14102.322,E2 -14102.322} C_VEL
LIN {X 0,Y 358.162,Z 181.496,A -85,B 0,C 180,E1 -14102.463,E2 -14102.463} C_VEL
LIN {X 0,Y 355.58,Z 276.806,A -85,B 0,C 180,E1 -14104.422,E2 -14104.422} C_VEL
LIN {X 0,Y 354.564,Z 291.192,A -85,B 0,C 180,E1 -14104.932,E2 -14104.932} C_VEL
LIN {X 0,Y 353.141,Z 305.581,A -85,B 0,C 180,E1 -14105.688,E2 -14105.688} C_VEL
LIN {X 0,Y 351.615,Z 318.392,A -85,B 0,C 180,E1 -14106.597,E2 -14106.597} C_VEL
LIN {X 0,Y 349.944,Z 330.777,A -85,B 0,C 180,E1 -14107.724,E2 -14107.724} C_VEL
LIN {X 0,Y 347.953,Z 343.325,A -85,B 0,C 180,E1 -14109.146,E2 -14109.146} C_VEL
LIN {X 0,Y 346.06,Z 354.534,A -85,B 0,C 180,E1 -14110.73,E2 -14110.73} C_VEL
LIN {X 0,Y 344.252,Z 364.583,A -85,B 0,C 180,E1 -14112.475,E2 -14112.475} C_VEL
LIN {X 0,Y 342.762,Z 372.945,A -85,B 0,C 180,E1 -14114.236,E2 -14114.236} C_VEL
LIN {X 0,Y 341.509,Z 380.951,A -85,B 0,C 180,E1 -14116.31,E2 -14116.31} C_VEL
LIN {X 0,Y 340.492,Z 386.609,A -85,B 0,C 180,E1 -14118.088,E2 -14118.088} C_VEL
LIN {X 0,Y 339.7,Z 392.548,A -85,B 0,C 180,E1 -14120.473,E2 -14120.473} C_VEL
LIN {X 0,Y 339.246,Z 396.925,A -85,B 0,C 180,E1 -14122.86,E2 -14122.86} C_VEL
LIN {X 0,Y 339.043,Z 399.868,A -85,B 0,C 180,E1 -14125.244,E2 -14125.244} C_VEL
LIN {X 0,Y 338.981,Z 401.453,A -85,B 0,C 180,E1 -14127.623,E2 -14127.623} C_VEL
LIN {X 0,Y 339.015,Z 401.708,A -85,B 0,C 180,E1 -14130,E2 -14130} C_VEL
LIN {X 0,Y 338.99,Z 400.628,A -85,B 0,C 180,E1 -14132.376,E2 -14132.376} C_VEL
LIN {X 0,Y 339.048,Z 399.583,A -85,B 0,C 180,E1 -14133.565,E2 -14133.565} C_VEL
LIN {X 0,Y 339.087,Z 396.441,A -85,B 0,C 180,E1 -14135.948,E2 -14135.948} C_VEL
LIN {X 0,Y 339.335,Z 391.794,A -85,B 0,C 180,E1 -14138.336,E2 -14138.336} C_VEL
LIN {X 0,Y 339.695,Z 387.219,A -85,B 0,C 180,E1 -14140.128,E2 -14140.128} C_VEL
LIN {X 0,Y 340.421,Z 380.615,A -85,B 0,C 180,E1 -14142.217,E2 -14142.217} C_VEL
LIN {X 0,Y 341.354,Z 372.403,A -85,B 0,C 180,E1 -14144.304,E2 -14144.304} C_VEL
LIN {X 0,Y 342.379,Z 363.793,A -85,B 0,C 180,E1 -14146.088,E2 -14146.088} C_VEL
LIN {X 0,Y 343.776,Z 353.357,A -85,B 0,C 180,E1 -14147.857,E2 -14147.857} C_VEL
LIN {X 0,Y 345.056,Z 344.032,A -85,B 0,C 180,E1 -14149.173,E2 -14149.173} C_VEL
LIN {X 0,Y 346.501,Z 332.868,A -85,B 0,C 180,E1 -14150.48,E2 -14150.48} C_VEL
LIN {X 0,Y 347.831,Z 320.542,A -85,B 0,C 180,E1 -14151.652,E2 -14151.652} C_VEL
LIN {X 0,Y 349.079,Z 307.2,A -85,B 0,C 180,E1 -14152.646,E2 -14152.646} C_VEL
LIN {X 0,Y 350.27,Z 293.115,A -85,B 0,C 180,E1 -14153.423,E2 -14153.423} C_VEL
LIN {X 0,Y 351.16,Z 278.253,A -85,B 0,C 180,E1 -14153.987,E2 -14153.987} C_VEL
LIN {X 0,Y 351.845,Z 253.688,A -85,B 0,C 180,E1 -14154.525,E2 -14154.525} C_VEL
LIN {X 0,Y 353.357,Z 178.213,A -85,B 0,C 180,E1 -14156.057,E2 -14156.057} C_VEL
LIN {X 0,Y 347.704,Z 144.701,A -85,B 0,C 180,E1 -14157.208,E2 -14157.208} C_VEL
LIN {X 0,Y 345.652,Z 138.445,A -85,B 0,C 180,E1 -14157.52,E2 -14157.52} C_VEL
LIN {X 0,Y 342.895,Z 125.407,A -85,B 0,C 180,E1 -14160.824,E2 -14160.824} C_VEL
LIN {X 0,Y 340.71,Z 116.171,A -85,B 0,C 180,E1 -14163.312,E2 -14163.312} C_VEL
LIN {X 0,Y 340.704,Z 116.17,A -85,B 0,C 180,E1 -14166.741,E2 -14166.741} C_VEL
LIN {X 0,Y 340.687,Z 116.173,A -85,B 0,C 180,E1 -14170.247,E2 -14170.247} C_VEL
LIN {X 0,Y 340.676,Z 116.177,A -85,B 0,C 180,E1 -14173.777,E2 -14173.777} C_VEL
LIN {X 0,Y 340.74,Z 116.163,A -85,B 0,C 180,E1 -14177.106,E2 -14177.106} C_VEL
LIN {X 0,Y 340.732,Z 116.162,A -85,B 0,C 180,E1 -14180.252,E2 -14180.252} C_VEL
LIN {X 0,Y 340.709,Z 116.171,A -85,B 0,C 180,E1 -14183.559,E2 -14183.559} C_VEL
LIN {X 0,Y 340.691,Z 116.168,A -85,B 0,C 180,E1 -14186.153,E2 -14186.153} C_VEL
LIN {X 0,Y 340.773,Z 116.158,A -85,B 0,C 180,E1 -14190.332,E2 -14190.332} C_VEL
LIN {X 0,Y 340.803,Z 116.159,A -85,B 0,C 180,E1 -14193.02,E2 -14193.02} C_VEL
LIN {X 0,Y 340.727,Z 116.167,A -85,B 0,C 180,E1 -14196.927,E2 -14196.927} C_VEL
LIN {X 0,Y 340.789,Z 116.16,A -85,B 0,C 180,E1 -14200.734,E2 -14200.734} C_VEL
LIN {X 0,Y 340.786,Z 116.16,A -85,B 0,C 180,E1 -14203.219,E2 -14203.219} C_VEL
LIN {X 0,Y 340.843,Z 116.152,A -85,B 0,C 180,E1 -14206.891,E2 -14206.891} C_VEL
LIN {X 0,Y 340.923,Z 116.145,A -85,B 0,C 180,E1 -14210.508,E2 -14210.508} C_VEL
LIN {X 0,Y 341.058,Z 116.124,A -85,B 0,C 180,E1 -14212.898,E2 -14212.898} C_VEL
LIN {X 0,Y 341.167,Z 116.11,A -85,B 0,C 180,E1 -14217.639,E2 -14217.639} C_VEL
LIN {X 0,Y 341.294,Z 116.096,A -85,B 0,C 180,E1 -14220,E2 -14220} C_VEL
LIN {X 0,Y 341.167,Z 116.112,A -85,B 0,C 180,E1 -14222.361,E2 -14222.361} C_VEL
LIN {X 0,Y 341.017,Z 116.128,A -85,B 0,C 180,E1 -14227.103,E2 -14227.103} C_VEL
LIN {X 0,Y 340.87,Z 116.145,A -85,B 0,C 180,E1 -14230.694,E2 -14230.694} C_VEL
LIN {X 0,Y 340.862,Z 116.149,A -85,B 0,C 180,E1 -14234.325,E2 -14234.325} C_VEL
LIN {X 0,Y 340.836,Z 116.149,A -85,B 0,C 180,E1 -14238.467,E2 -14238.467} C_VEL
LIN {X 0,Y 340.753,Z 116.164,A -85,B 0,C 180,E1 -14241.857,E2 -14241.857} C_VEL
LIN {X 0,Y 340.772,Z 116.162,A -85,B 0,C 180,E1 -14245.665,E2 -14245.665} C_VEL
LIN {X 0,Y 340.728,Z 116.165,A -85,B 0,C 180,E1 -14248.321,E2 -14248.321} C_VEL
LIN {X 0,Y 340.697,Z 116.171,A -85,B 0,C 180,E1 -14251.045,E2 -14251.045} C_VEL
LIN {X 0,Y 340.718,Z 116.169,A -85,B 0,C 180,E1 -14255.279,E2 -14255.279} C_VEL
LIN {X 0,Y 340.709,Z 116.167,A -85,B 0,C 180,E1 -14258.386,E2 -14258.386} C_VEL
LIN {X 0,Y 340.699,Z 116.167,A -85,B 0,C 180,E1 -14262.046,E2 -14262.046} C_VEL
LIN {X 0,Y 340.682,Z 116.17,A -85,B 0,C 180,E1 -14265.462,E2 -14265.462} C_VEL
LIN {X 0,Y 340.686,Z 116.174,A -85,B 0,C 180,E1 -14268.691,E2 -14268.691} C_VEL
LIN {X 0,Y 340.733,Z 116.161,A -85,B 0,C 180,E1 -14271.773,E2 -14271.773} C_VEL
LIN {X 0,Y 340.724,Z 116.165,A -85,B 0,C 180,E1 -14275.596,E2 -14275.596} C_VEL
LIN {X 0,Y 340.696,Z 116.17,A -85,B 0,C 180,E1 -14278.955,E2 -14278.955} C_VEL
LIN {X 0,Y 340.722,Z 116.165,A -85,B 0,C 180,E1 -14283.013,E2 -14283.013} C_VEL
LIN {X 0,Y 340.769,Z 116.214,A -85,B 0,C 180,E1 -14285.883,E2 -14285.883} C_VEL
LIN {X 0,Y 342.775,Z 125.107,A -85,B 0,C 180,E1 -14288.343,E2 -14288.343} C_VEL
LIN {X 0,Y 350.721,Z 145.003,A -85,B 0,C 180,E1 -14289.399,E2 -14289.399} C_VEL
LIN {X 0,Y 352.438,Z 150.772,A -85,B 0,C 180,E1 -14289.652,E2 -14289.652} C_VEL
LIN {X 0,Y 353.858,Z 158.628,A -85,B 0,C 180,E1 -14289.927,E2 -14289.927} C_VEL
LIN {X 0,Y 351.514,Z 261.347,A -85,B 0,C 180,E1 -14292.022,E2 -14292.022} C_VEL
LIN {X 0,Y 350.893,Z 275.912,A -85,B 0,C 180,E1 -14292.554,E2 -14292.554} C_VEL
LIN {X 0,Y 349.897,Z 289.831,A -85,B 0,C 180,E1 -14293.293,E2 -14293.293} C_VEL
LIN {X 0,Y 348.727,Z 302.77,A -85,B 0,C 180,E1 -14294.213,E2 -14294.213} C_VEL
LIN {X 0,Y 347.43,Z 315.299,A -85,B 0,C 180,E1 -14295.354,E2 -14295.354} C_VEL
LIN {X 0,Y 346.056,Z 326.726,A -85,B 0,C 180,E1 -14296.644,E2 -14296.644} C_VEL
LIN {X 0,Y 344.497,Z 338.193,A -85,B 0,C 180,E1 -14298.229,E2 -14298.229} C_VEL
LIN {X 0,Y 343.237,Z 348.44,A -85,B 0,C 180,E1 -14299.977,E2 -14299.977} C_VEL
LIN {X 0,Y 342.008,Z 356.919,A -85,B 0,C 180,E1 -14301.73,E2 -14301.73} C_VEL
LIN {X 0,Y 340.98,Z 365.031,A -85,B 0,C 180,E1 -14303.788,E2 -14303.788} C_VEL
LIN {X 0,Y 340.14,Z 371.571,A -85,B 0,C 180,E1 -14305.853,E2 -14305.853} C_VEL
LIN {X 0,Y 339.549,Z 377.383,A -85,B 0,C 180,E1 -14308.221,E2 -14308.221} C_VEL
LIN {X 0,Y 339.285,Z 380.752,A -85,B 0,C 180,E1 -14310,E2 -14310} C_VEL
LIN {X 0,Y 339.042,Z 383.926,A -85,B 0,C 180,E1 -14312.376,E2 -14312.376} C_VEL
LIN {X 0,Y 339.047,Z 385.731,A -85,B 0,C 180,E1 -14314.756,E2 -14314.756} C_VEL
LIN {X 0,Y 339.095,Z 386.138,A -85,B 0,C 180,E1 -14315.948,E2 -14315.948} C_VEL
LIN {X 0,Y 338.989,Z 385.966,A -85,B 0,C 180,E1 -14318.345,E2 -14318.345} C_VEL
LIN {X 0,Y 339.113,Z 384.455,A -85,B 0,C 180,E1 -14320.75,E2 -14320.75} C_VEL
LIN {X 0,Y 339.626,Z 381.563,A -85,B 0,C 180,E1 -14323.158,E2 -14323.158} C_VEL
LIN {X 0,Y 340.206,Z 377.206,A -85,B 0,C 180,E1 -14325.578,E2 -14325.578} C_VEL
LIN {X 0,Y 340.937,Z 372.859,A -85,B 0,C 180,E1 -14327.392,E2 -14327.392} C_VEL
LIN {X 0,Y 342.057,Z 366.51,A -85,B 0,C 180,E1 -14329.504,E2 -14329.504} C_VEL
LIN {X 0,Y 343.454,Z 358.574,A -85,B 0,C 180,E1 -14331.613,E2 -14331.613} C_VEL
LIN {X 0,Y 345.062,Z 350.092,A -85,B 0,C 180,E1 -14333.434,E2 -14333.434} C_VEL
LIN {X 0,Y 346.765,Z 340.169,A -85,B 0,C 180,E1 -14335.19,E2 -14335.19} C_VEL
LIN {X 0,Y 348.667,Z 328.907,A -85,B 0,C 180,E1 -14336.809,E2 -14336.809} C_VEL
LIN {X 0,Y 350.618,Z 316.625,A -85,B 0,C 180,E1 -14338.218,E2 -14338.218} C_VEL
LIN {X 0,Y 352.084,Z 305.317,A -85,B 0,C 180,E1 -14339.278,E2 -14339.278} C_VEL
LIN {X 0,Y 352.36,Z 303.512,A -85,B 0,C 180,E1 -14339.419,E2 -14339.419} C_VEL
LIN {X 0,Y 352.5,Z 298.316,A -85,B 0,C 180,E1 -14339.861,E2 -14339.861} C_VEL
LIN {X 0,Y 350.917,Z 289.754,A -85,B 0,C 180,E1 -14340.642,E2 -14340.642} C_VEL
LIN {X 0,Y 349.107,Z 281.033,A -85,B 0,C 180,E1 -14341.36,E2 -14341.36} C_VEL
LIN {X 0,Y 348.824,Z 275.481,A -85,B 0,C 180,E1 -14341.683,E2 -14341.683} C_VEL
LIN {X 0,Y 349.646,Z 261.626,A -85,B 0,C 180,E1 -14342.178,E2 -14342.178} C_VEL
LIN {X 0,Y 352.487,Z 161.67,A -85,B 0,C 180,E1 -14344.254,E2 -14344.254} C_VEL
LIN {X 0,Y 349.832,Z 154.778,A -85,B 0,C 180,E1 -14344.675,E2 -14344.675} C_VEL
LIN {X 0,Y 341.363,Z 136.372,A -85,B 0,C 180,E1 -14345.991,E2 -14345.991} C_VEL
LIN {X 0,Y 335.839,Z 125.352,A -85,B 0,C 180,E1 -14346.877,E2 -14346.877} C_VEL
LIN {X 0,Y 333.624,Z 117.053,A -85,B 0,C 180,E1 -14349.635,E2 -14349.635} C_VEL
LIN {X 0,Y 333.628,Z 117.053,A -85,B 0,C 180,E1 -14352.498,E2 -14352.498} C_VEL
LIN {X 0,Y 333.594,Z 117.044,A -85,B 0,C 180,E1 -14355.954,E2 -14355.954} C_VEL
LIN {X 0,Y 333.603,Z 117.041,A -85,B 0,C 180,E1 -14359.324,E2 -14359.324} C_VEL
LIN {X 0,Y 333.662,Z 117.048,A -85,B 0,C 180,E1 -14363.169,E2 -14363.169} C_VEL
LIN {X 0,Y 333.674,Z 117.049,A -85,B 0,C 180,E1 -14365.341,E2 -14365.341} C_VEL
LIN {X 0,Y 333.63,Z 117.051,A -85,B 0,C 180,E1 -14368.222,E2 -14368.222} C_VEL
LIN {X 0,Y 333.655,Z 117.045,A -85,B 0,C 180,E1 -14371.022,E2 -14371.022} C_VEL
LIN {X 0,Y 333.697,Z 117.044,A -85,B 0,C 180,E1 -14375.088,E2 -14375.088} C_VEL
LIN {X 0,Y 333.668,Z 117.047,A -85,B 0,C 180,E1 -14379.018,E2 -14379.018} C_VEL
LIN {X 0,Y 333.743,Z 117.028,A -85,B 0,C 180,E1 -14381.586,E2 -14381.586} C_VEL
LIN {X 0,Y 333.809,Z 117.024,A -85,B 0,C 180,E1 -14385.577,E2 -14385.577} C_VEL
LIN {X 0,Y 333.834,Z 117.025,A -85,B 0,C 180,E1 -14389.078,E2 -14389.078} C_VEL
LIN {X 0,Y 333.965,Z 117.01,A -85,B 0,C 180,E1 -14392.746,E2 -14392.746} C_VEL
LIN {X 0,Y 333.799,Z 117.025,A -85,B 0,C 180,E1 -14395.169,E2 -14395.169} C_VEL
LIN {X 0,Y 334.102,Z 116.988,A -85,B 0,C 180,E1 -14397.589,E2 -14397.589} C_VEL
LIN {X 0,Y 334.226,Z 116.972,A -85,B 0,C 180,E1 -14400,E2 -14400} C_VEL
LIN {X 0,Y 334.102,Z 116.989,A -85,B 0,C 180,E1 -14402.411,E2 -14402.411} C_VEL
LIN {X 0,Y 333.992,Z 116.995,A -85,B 0,C 180,E1 -14406.039,E2 -14406.039} C_VEL
LIN {X 0,Y 333.821,Z 117.026,A -85,B 0,C 180,E1 -14409.696,E2 -14409.696} C_VEL
LIN {X 0,Y 333.797,Z 117.031,A -85,B 0,C 180,E1 -14413.391,E2 -14413.391} C_VEL
LIN {X 0,Y 333.747,Z 117.027,A -85,B 0,C 180,E1 -14417.146,E2 -14417.146} C_VEL
LIN {X 0,Y 333.737,Z 117.031,A -85,B 0,C 180,E1 -14419.69,E2 -14419.69} C_VEL
LIN {X 0,Y 333.693,Z 117.039,A -85,B 0,C 180,E1 -14422.278,E2 -14422.278} C_VEL
LIN {X 0,Y 333.736,Z 117.033,A -85,B 0,C 180,E1 -14426.246,E2 -14426.246} C_VEL
LIN {X 0,Y 333.711,Z 117.034,A -85,B 0,C 180,E1 -14428.972,E2 -14428.972} C_VEL
LIN {X 0,Y 333.644,Z 117.044,A -85,B 0,C 180,E1 -14432.587,E2 -14432.587} C_VEL
LIN {X 0,Y 333.676,Z 117.041,A -85,B 0,C 180,E1 -14436.139,E2 -14436.139} C_VEL
LIN {X 0,Y 333.646,Z 117.031,A -85,B 0,C 180,E1 -14439.192,E2 -14439.192} C_VEL
LIN {X 0,Y 333.633,Z 117.052,A -85,B 0,C 180,E1 -14442.5,E2 -14442.5} C_VEL
LIN {X 0,Y 333.597,Z 117.052,A -85,B 0,C 180,E1 -14445.955,E2 -14445.955} C_VEL
LIN {X 0,Y 333.648,Z 117.047,A -85,B 0,C 180,E1 -14449.315,E2 -14449.315} C_VEL
LIN {X 0,Y 333.681,Z 117.103,A -85,B 0,C 180,E1 -14453.315,E2 -14453.315} C_VEL
LIN {X 0,Y 336.582,Z 127.96,A -85,B 0,C 180,E1 -14456.639,E2 -14456.639} C_VEL
LIN {X 0,Y 339.013,Z 138.063,A -85,B 0,C 180,E1 -14459.525,E2 -14459.525} C_VEL
LIN {X 0,Y 346.805,Z 155.263,A -85,B 0,C 180,E1 -14460.761,E2 -14460.761} C_VEL
LIN {X 0,Y 350.815,Z 174.851,A -85,B 0,C 180,E1 -14461.619,E2 -14461.619} C_VEL
LIN {X 0,Y 351.999,Z 182.159,A -85,B 0,C 180,E1 -14461.903,E2 -14461.903} C_VEL
LIN {X 0,Y 349.374,Z 275.886,A -85,B 0,C 180,E1 -14463.853,E2 -14463.853} C_VEL
LIN {X 0,Y 348.308,Z 290.534,A -85,B 0,C 180,E1 -14464.37,E2 -14464.37} C_VEL
LIN {X 0,Y 346.962,Z 303.926,A -85,B 0,C 180,E1 -14465.066,E2 -14465.066} C_VEL
LIN {X 0,Y 345.352,Z 317.014,A -85,B 0,C 180,E1 -14465.983,E2 -14465.983} C_VEL
LIN {X 0,Y 343.626,Z 329.671,A -85,B 0,C 180,E1 -14467.133,E2 -14467.133} C_VEL
LIN {X 0,Y 341.76,Z 341.214,A -85,B 0,C 180,E1 -14468.433,E2 -14468.433} C_VEL
LIN {X 0,Y 340.036,Z 350.84,A -85,B 0,C 180,E1 -14469.745,E2 -14469.745} C_VEL
LIN {X 0,Y 338.065,Z 361.526,A -85,B 0,C 180,E1 -14471.516,E2 -14471.516} C_VEL
LIN {X 0,Y 336.367,Z 370.365,A -85,B 0,C 180,E1 -14473.304,E2 -14473.304} C_VEL
LIN {X 0,Y 335.042,Z 377.838,A -85,B 0,C 180,E1 -14475.139,E2 -14475.139} C_VEL
LIN {X 0,Y 333.875,Z 384.801,A -85,B 0,C 180,E1 -14477.231,E2 -14477.231} C_VEL
LIN {X 0,Y 332.832,Z 391.166,A -85,B 0,C 180,E1 -14479.66,E2 -14479.66} C_VEL
LIN {X 0,Y 332.363,Z 394.846,A -85,B 0,C 180,E1 -14481.488,E2 -14481.488} C_VEL
LIN {X 0,Y 332.041,Z 398.465,A -85,B 0,C 180,E1 -14483.925,E2 -14483.925} C_VEL
LIN {X 0,Y 331.945,Z 400.698,A -85,B 0,C 180,E1 -14486.358,E2 -14486.358} C_VEL
LIN {X 0,Y 331.884,Z 401.59,A -85,B 0,C 180,E1 -14488.786,E2 -14488.786} C_VEL
LIN {X 0,Y 331.899,Z 401.153,A -85,B 0,C 180,E1 -14491.213,E2 -14491.213} C_VEL
LIN {X 0,Y 331.951,Z 399.375,A -85,B 0,C 180,E1 -14493.641,E2 -14493.641} C_VEL
LIN {X 0,Y 331.998,Z 396.204,A -85,B 0,C 180,E1 -14496.076,E2 -14496.076} C_VEL
LIN {X 0,Y 332.28,Z 391.514,A -85,B 0,C 180,E1 -14498.514,E2 -14498.514} C_VEL
LIN {X 0,Y 332.662,Z 386.923,A -85,B 0,C 180,E1 -14500.345,E2 -14500.345} C_VEL
LIN {X 0,Y 333.436,Z 380.285,A -85,B 0,C 180,E1 -14502.477,E2 -14502.477} C_VEL
LIN {X 0,Y 334.376,Z 372.017,A -85,B 0,C 180,E1 -14504.609,E2 -14504.609} C_VEL
LIN {X 0,Y 335.524,Z 363.366,A -85,B 0,C 180,E1 -14506.426,E2 -14506.426} C_VEL
LIN {X 0,Y 336.947,Z 352.867,A -85,B 0,C 180,E1 -14508.232,E2 -14508.232} C_VEL
LIN {X 0,Y 338.447,Z 342.306,A -85,B 0,C 180,E1 -14509.721,E2 -14509.721} C_VEL
LIN {X 0,Y 339.957,Z 330.8,A -85,B 0,C 180,E1 -14511.051,E2 -14511.051} C_VEL
LIN {X 0,Y 341.338,Z 318.797,A -85,B 0,C 180,E1 -14512.174,E2 -14512.174} C_VEL
LIN {X 0,Y 342.628,Z 305.144,A -85,B 0,C 180,E1 -14513.177,E2 -14513.177} C_VEL
LIN {X 0,Y 343.812,Z 291.168,A -85,B 0,C 180,E1 -14513.931,E2 -14513.931} C_VEL
LIN {X 0,Y 344.653,Z 276.56,A -85,B 0,C 180,E1 -14514.469,E2 -14514.469} C_VEL
LIN {X 0,Y 346.891,Z 179.432,A -85,B 0,C 180,E1 -14516.496,E2 -14516.496} C_VEL
LIN {X 0,Y 341.415,Z 146.568,A -85,B 0,C 180,E1 -14517.651,E2 -14517.651} C_VEL
LIN {X 0,Y 338.433,Z 138.236,A -85,B 0,C 180,E1 -14518.103,E2 -14518.103} C_VEL
LIN {X 0,Y 335.542,Z 124.941,A -85,B 0,C 180,E1 -14521.576,E2 -14521.576} C_VEL
LIN {X 0,Y 333.679,Z 117.049,A -85,B 0,C 180,E1 -14523.746,E2 -14523.746} C_VEL
LIN {X 0,Y 333.651,Z 117.051,A -85,B 0,C 180,E1 -14527.651,E2 -14527.651} C_VEL
LIN {X 0,Y 333.645,Z 117.047,A -85,B 0,C 180,E1 -14530.767,E2 -14530.767} C_VEL
LIN {X 0,Y 333.642,Z 117.049,A -85,B 0,C 180,E1 -14534.259,E2 -14534.259} C_VEL
LIN {X 0,Y 333.695,Z 117.045,A -85,B 0,C 180,E1 -14537.627,E2 -14537.627} C_VEL
LIN {X 0,Y 333.677,Z 117.041,A -85,B 0,C 180,E1 -14541.196,E2 -14541.196} C_VEL
LIN {X 0,Y 333.684,Z 117.046,A -85,B 0,C 180,E1 -14545.226,E2 -14545.226} C_VEL
LIN {X 0,Y 333.696,Z 117.042,A -85,B 0,C 180,E1 -14549.638,E2 -14549.638} C_VEL
LIN {X 0,Y 333.742,Z 117.035,A -85,B 0,C 180,E1 -14552.401,E2 -14552.401} C_VEL
LIN {X 0,Y 333.726,Z 117.04,A -85,B 0,C 180,E1 -14555.091,E2 -14555.091} C_VEL
LIN {X 0,Y 333.684,Z 117.047,A -85,B 0,C 180,E1 -14559.02,E2 -14559.02} C_VEL
LIN {X 0,Y 333.792,Z 117.027,A -85,B 0,C 180,E1 -14561.59,E2 -14561.59} C_VEL
LIN {X 0,Y 333.807,Z 117.026,A -85,B 0,C 180,E1 -14565.577,E2 -14565.577} C_VEL
LIN {X 0,Y 333.833,Z 117.025,A -85,B 0,C 180,E1 -14569.078,E2 -14569.078} C_VEL
LIN {X 0,Y 334.005,Z 117.004,A -85,B 0,C 180,E1 -14572.747,E2 -14572.747} C_VEL
LIN {X 0,Y 333.807,Z 117.025,A -85,B 0,C 180,E1 -14575.169,E2 -14575.169} C_VEL
LIN {X 0,Y 334.104,Z 116.99,A -85,B 0,C 180,E1 -14577.589,E2 -14577.589} C_VEL
LIN {X 0,Y 334.245,Z 116.974,A -85,B 0,C 180,E1 -14580,E2 -14580} C_VEL
LIN {X 0,Y 334.104,Z 116.991,A -85,B 0,C 180,E1 -14582.411,E2 -14582.411} C_VEL
LIN {X 0,Y 333.97,Z 117.007,A -85,B 0,C 180,E1 -14586.51,E2 -14586.51} C_VEL
LIN {X 0,Y 333.849,Z 117.022,A -85,B 0,C 180,E1 -14589.696,E2 -14589.696} C_VEL
LIN {X 0,Y 333.796,Z 117.029,A -85,B 0,C 180,E1 -14593.392,E2 -14593.392} C_VEL
LIN {X 0,Y 333.746,Z 117.033,A -85,B 0,C 180,E1 -14597.147,E2 -14597.147} C_VEL
LIN {X 0,Y 333.738,Z 117.039,A -85,B 0,C 180,E1 -14599.691,E2 -14599.691} C_VEL
LIN {X 0,Y 333.692,Z 117.041,A -85,B 0,C 180,E1 -14602.278,E2 -14602.278} C_VEL
LIN {X 0,Y 333.735,Z 117.035,A -85,B 0,C 180,E1 -14606.247,E2 -14606.247} C_VEL
LIN {X 0,Y 333.69,Z 117.044,A -85,B 0,C 180,E1 -14608.974,E2 -14608.974} C_VEL
LIN {X 0,Y 333.643,Z 117.046,A -85,B 0,C 180,E1 -14612.587,E2 -14612.587} C_VEL
LIN {X 0,Y 333.676,Z 117.042,A -85,B 0,C 180,E1 -14616.139,E2 -14616.139} C_VEL
LIN {X 0,Y 333.646,Z 117.051,A -85,B 0,C 180,E1 -14619.193,E2 -14619.193} C_VEL
LIN {X 0,Y 333.634,Z 117.048,A -85,B 0,C 180,E1 -14622.501,E2 -14622.501} C_VEL
LIN {X 0,Y 333.62,Z 117.049,A -85,B 0,C 180,E1 -14625.959,E2 -14625.959} C_VEL
LIN {X 0,Y 333.647,Z 117.046,A -85,B 0,C 180,E1 -14629.316,E2 -14629.316} C_VEL
LIN {X 0,Y 333.665,Z 117.046,A -85,B 0,C 180,E1 -14633.168,E2 -14633.168} C_VEL
LIN {X 0,Y 333.675,Z 117.043,A -85,B 0,C 180,E1 -14635.342,E2 -14635.342} C_VEL
LIN {X 0,Y 333.631,Z 117.053,A -85,B 0,C 180,E1 -14638.222,E2 -14638.222} C_VEL
LIN {X 0,Y 333.656,Z 117.047,A -85,B 0,C 180,E1 -14641.023,E2 -14641.023} C_VEL
LIN {X 0,Y 333.698,Z 117.041,A -85,B 0,C 180,E1 -14645.089,E2 -14645.089} C_VEL
LIN {X 0,Y 333.725,Z 117.172,A -85,B 0,C 180,E1 -14645.464,E2 -14645.464} C_VEL
LIN {X 0,Y 335.561,Z 125.149,A -85,B 0,C 180,E1 -14647.756,E2 -14647.756} C_VEL
LIN {X 0,Y 343.776,Z 145.488,A -85,B 0,C 180,E1 -14648.883,E2 -14648.883} C_VEL
LIN {X 0,Y 345.975,Z 151.96,A -85,B 0,C 180,E1 -14649.198,E2 -14649.198} C_VEL
LIN {X 0,Y 347.342,Z 158.921,A -85,B 0,C 180,E1 -14649.456,E2 -14649.456} C_VEL
LIN {X 0,Y 344.941,Z 261.588,A -85,B 0,C 180,E1 -14651.591,E2 -14651.591} C_VEL
LIN {X 0,Y 344.284,Z 276.127,A -85,B 0,C 180,E1 -14652.131,E2 -14652.131} C_VEL
LIN {X 0,Y 343.268,Z 290.031,A -85,B 0,C 180,E1 -14652.884,E2 -14652.884} C_VEL
LIN {X 0,Y 341.953,Z 303.842,A -85,B 0,C 180,E1 -14653.892,E2 -14653.892} C_VEL
LIN {X 0,Y 340.61,Z 316.197,A -85,B 0,C 180,E1 -14655.054,E2 -14655.054} C_VEL
LIN {X 0,Y 339.071,Z 328.655,A -85,B 0,C 180,E1 -14656.516,E2 -14656.516} C_VEL
LIN {X 0,Y 337.585,Z 338.861,A -85,B 0,C 180,E1 -14657.984,E2 -14657.984} C_VEL
LIN {X 0,Y 336.288,Z 349.003,A -85,B 0,C 180,E1 -14659.768,E2 -14659.768} C_VEL
LIN {X 0,Y 335.011,Z 357.419,A -85,B 0,C 180,E1 -14661.556,E2 -14661.556} C_VEL
LIN {X 0,Y 333.952,Z 365.454,A -85,B 0,C 180,E1 -14663.657,E2 -14663.657} C_VEL
LIN {X 0,Y 333.092,Z 371.943,A -85,B 0,C 180,E1 -14665.765,E2 -14665.765} C_VEL
LIN {X 0,Y 332.482,Z 377.707,A -85,B 0,C 180,E1 -14668.183,E2 -14668.183} C_VEL
LIN {X 0,Y 332.186,Z 381.038,A -85,B 0,C 180,E1 -14670,E2 -14670} C_VEL
LIN {X 0,Y 331.956,Z 384.162,A -85,B 0,C 180,E1 -14672.427,E2 -14672.427} C_VEL
LIN {X 0,Y 331.953,Z 385.926,A -85,B 0,C 180,E1 -14674.858,E2 -14674.858} C_VEL
LIN {X 0,Y 331.991,Z 386.312,A -85,B 0,C 180,E1 -14676.076,E2 -14676.076} C_VEL
LIN {X 0,Y 331.909,Z 386.098,A -85,B 0,C 180,E1 -14678.524,E2 -14678.524} C_VEL
LIN {X 0,Y 332.071,Z 384.545,A -85,B 0,C 180,E1 -14680.981,E2 -14680.981} C_VEL
LIN {X 0,Y 332.632,Z 381.364,A -85,B 0,C 180,E1 -14683.611,E2 -14683.611} C_VEL
LIN {X 0,Y 333.223,Z 377.207,A -85,B 0,C 180,E1 -14685.913,E2 -14685.913} C_VEL
LIN {X 0,Y 334.013,Z 372.81,A -85,B 0,C 180,E1 -14687.764,E2 -14687.764} C_VEL
LIN {X 0,Y 335.236,Z 366.408,A -85,B 0,C 180,E1 -14689.918,E2 -14689.918} C_VEL
LIN {X 0,Y 336.721,Z 358.414,A -85,B 0,C 180,E1 -14692.067,E2 -14692.067} C_VEL
LIN {X 0,Y 338.483,Z 349.512,A -85,B 0,C 180,E1 -14693.994,E2 -14693.994} C_VEL
LIN {X 0,Y 340.205,Z 339.865,A -85,B 0,C 180,E1 -14695.71,E2 -14695.71} C_VEL
LIN {X 0,Y 342.25,Z 328.461,A -85,B 0,C 180,E1 -14697.353,E2 -14697.353} C_VEL
LIN {X 0,Y 344.16,Z 316.666,A -85,B 0,C 180,E1 -14698.724,E2 -14698.724} C_VEL
LIN {X 0,Y 345.852,Z 304.56,A -85,B 0,C 180,E1 -14699.859,E2 -14699.859} C_VEL
LIN {X 0,Y 347.363,Z 291.707,A -85,B 0,C 180,E1 -14700.806,E2 -14700.806} C_VEL
LIN {X 0,Y 348.654,Z 277.168,A -85,B 0,C 180,E1 -14701.608,E2 -14701.608} C_VEL
LIN {X 0,Y 348.824,Z 275.481,A -85,B 0,C 180,E1 -14701.683,E2 -14701.683} C_VEL
LIN {X 0,Y 348.571,Z 269.841,A -85,B 0,C 180,E1 -14701.976,E2 -14701.976} C_VEL
LIN {X 0,Y 346.493,Z 260.652,A -85,B 0,C 180,E1 -14702.493,E2 -14702.493} C_VEL
LIN {X 0,Y 344.341,Z 251.358,A -85,B 0,C 180,E1 -14702.935,E2 -14702.935} C_VEL
LIN {X 0,Y 343.968,Z 245.558,A -85,B 0,C 180,E1 -14703.106,E2 -14703.106} C_VEL
LIN {X 0,Y 346.292,Z 162.935,A -85,B 0,C 180,E1 -14704.836,E2 -14704.836} C_VEL
LIN {X 0,Y 338.166,Z 144.51,A -85,B 0,C 180,E1 -14706.136,E2 -14706.136} C_VEL
LIN {X 0,Y 330.415,Z 129.054,A -85,B 0,C 180,E1 -14707.401,E2 -14707.401} C_VEL
LIN {X 0,Y 328.606,Z 125.495,A -85,B 0,C 180,E1 -14707.728,E2 -14707.728} C_VEL
LIN {X 0,Y 326.581,Z 117.93,A -85,B 0,C 180,E1 -14710.299,E2 -14710.299} C_VEL
LIN {X 0,Y 326.56,Z 117.933,A -85,B 0,C 180,E1 -14713.526,E2 -14713.526} C_VEL
LIN {X 0,Y 326.573,Z 117.927,A -85,B 0,C 180,E1 -14717.029,E2 -14717.029} C_VEL
LIN {X 0,Y 326.572,Z 117.913,A -85,B 0,C 180,E1 -14720.781,E2 -14720.781} C_VEL
LIN {X 0,Y 326.611,Z 117.921,A -85,B 0,C 180,E1 -14724.48,E2 -14724.48} C_VEL
LIN {X 0,Y 326.609,Z 117.923,A -85,B 0,C 180,E1 -14727.455,E2 -14727.455} C_VEL
LIN {X 0,Y 326.618,Z 117.918,A -85,B 0,C 180,E1 -14730.336,E2 -14730.336} C_VEL
LIN {X 0,Y 326.643,Z 117.917,A -85,B 0,C 180,E1 -14734.644,E2 -14734.644} C_VEL
LIN {X 0,Y 326.617,Z 117.919,A -85,B 0,C 180,E1 -14738.543,E2 -14738.543} C_VEL
LIN {X 0,Y 326.708,Z 117.905,A -85,B 0,C 180,E1 -14741.175,E2 -14741.175} C_VEL
LIN {X 0,Y 326.764,Z 117.901,A -85,B 0,C 180,E1 -14745.433,E2 -14745.433} C_VEL
LIN {X 0,Y 326.77,Z 117.906,A -85,B 0,C 180,E1 -14748.839,E2 -14748.839} C_VEL
LIN {X 0,Y 326.92,Z 117.885,A -85,B 0,C 180,E1 -14752.589,E2 -14752.589} C_VEL
LIN {X 0,Y 326.766,Z 117.901,A -85,B 0,C 180,E1 -14755.064,E2 -14755.064} C_VEL
LIN {X 0,Y 327.043,Z 117.867,A -85,B 0,C 180,E1 -14757.536,E2 -14757.536} C_VEL
LIN {X 0,Y 327.178,Z 117.849,A -85,B 0,C 180,E1 -14760,E2 -14760} C_VEL
LIN {X 0,Y 327.042,Z 117.868,A -85,B 0,C 180,E1 -14762.463,E2 -14762.463} C_VEL
LIN {X 0,Y 326.946,Z 117.872,A -85,B 0,C 180,E1 -14766.17,E2 -14766.17} C_VEL
LIN {X 0,Y 326.784,Z 117.9,A -85,B 0,C 180,E1 -14769.907,E2 -14769.907} C_VEL
LIN {X 0,Y 326.76,Z 117.909,A -85,B 0,C 180,E1 -14773.685,E2 -14773.685} C_VEL
LIN {X 0,Y 326.7,Z 117.91,A -85,B 0,C 180,E1 -14777.528,E2 -14777.528} C_VEL
LIN {X 0,Y 326.663,Z 117.91,A -85,B 0,C 180,E1 -14780.135,E2 -14780.135} C_VEL
LIN {X 0,Y 326.653,Z 117.914,A -85,B 0,C 180,E1 -14784.129,E2 -14784.129} C_VEL
LIN {X 0,Y 326.685,Z 117.916,A -85,B 0,C 180,E1 -14786.857,E2 -14786.857} C_VEL
LIN {X 0,Y 326.639,Z 117.923,A -85,B 0,C 180,E1 -14790.611,E2 -14790.611} C_VEL
LIN {X 0,Y 326.607,Z 117.926,A -85,B 0,C 180,E1 -14794.019,E2 -14794.019} C_VEL
LIN {X 0,Y 326.628,Z 117.924,A -85,B 0,C 180,E1 -14797.238,E2 -14797.238} C_VEL
LIN {X 0,Y 326.578,Z 117.92,A -85,B 0,C 180,E1 -14801.131,E2 -14801.131} C_VEL
LIN {X 0,Y 326.527,Z 117.921,A -85,B 0,C 180,E1 -14804.743,E2 -14804.743} C_VEL
LIN {X 0,Y 326.577,Z 117.931,A -85,B 0,C 180,E1 -14808.154,E2 -14808.154} C_VEL
LIN {X 0,Y 326.626,Z 117.92,A -85,B 0,C 180,E1 -14812.136,E2 -14812.136} C_VEL
LIN {X 0,Y 326.608,Z 117.947,A -85,B 0,C 180,E1 -14812.594,E2 -14812.594} C_VEL
LIN {X 0,Y 329.168,Z 127.197,A -85,B 0,C 180,E1 -14815.543,E2 -14815.543} C_VEL
LIN {X 0,Y 331.777,Z 137.871,A -85,B 0,C 180,E1 -14818.711,E2 -14818.711} C_VEL
LIN {X 0,Y 340.865,Z 157.622,A -85,B 0,C 180,E1 -14820.203,E2 -14820.203} C_VEL
LIN {X 0,Y 343.101,Z 167.778,A -85,B 0,C 180,E1 -14820.682,E2 -14820.682} C_VEL
LIN {X 0,Y 345.845,Z 182.584,A -85,B 0,C 180,E1 -14821.314,E2 -14821.314} C_VEL
LIN {X 0,Y 343.126,Z 276.148,A -85,B 0,C 180,E1 -14823.299,E2 -14823.299} C_VEL
LIN {X 0,Y 342.039,Z 290.643,A -85,B 0,C 180,E1 -14823.824,E2 -14823.824} C_VEL
LIN {X 0,Y 340.581,Z 304.526,A -85,B 0,C 180,E1 -14824.566,E2 -14824.566} C_VEL
LIN {X 0,Y 338.894,Z 317.45,A -85,B 0,C 180,E1 -14825.496,E2 -14825.496} C_VEL
LIN {X 0,Y 337.112,Z 329.989,A -85,B 0,C 180,E1 -14826.665,E2 -14826.665} C_VEL
LIN {X 0,Y 335.173,Z 341.446,A -85,B 0,C 180,E1 -14827.987,E2 -14827.987} C_VEL
LIN {X 0,Y 333.01,Z 352.949,A -85,B 0,C 180,E1 -14829.621,E2 -14829.621} C_VEL
LIN {X 0,Y 331.025,Z 363.254,A -85,B 0,C 180,E1 -14831.43,E2 -14831.43} C_VEL
LIN {X 0,Y 329.275,Z 371.779,A -85,B 0,C 180,E1 -14833.253,E2 -14833.253} C_VEL
LIN {X 0,Y 327.75,Z 379.95,A -85,B 0,C 180,E1 -14835.406,E2 -14835.406} C_VEL
LIN {X 0,Y 326.573,Z 386.55,A -85,B 0,C 180,E1 -14837.572,E2 -14837.572} C_VEL
LIN {X 0,Y 325.627,Z 392.425,A -85,B 0,C 180,E1 -14840.057,E2 -14840.057} C_VEL
LIN {X 0,Y 325.102,Z 396.744,A -85,B 0,C 180,E1 -14842.547,E2 -14842.547} C_VEL
LIN {X 0,Y 324.867,Z 399.633,A -85,B 0,C 180,E1 -14845.036,E2 -14845.036} C_VEL
LIN {X 0,Y 324.818,Z 401.167,A -85,B 0,C 180,E1 -14847.52,E2 -14847.52} C_VEL
LIN {X 0,Y 324.826,Z 401.369,A -85,B 0,C 180,E1 -14850,E2 -14850} C_VEL
LIN {X 0,Y 324.826,Z 400.238,A -85,B 0,C 180,E1 -14852.48,E2 -14852.48} C_VEL
LIN {X 0,Y 324.853,Z 397.744,A -85,B 0,C 180,E1 -14854.964,E2 -14854.964} C_VEL
LIN {X 0,Y 325.034,Z 393.798,A -85,B 0,C 180,E1 -14857.454,E2 -14857.454} C_VEL
LIN {X 0,Y 325.337,Z 389.793,A -85,B 0,C 180,E1 -14859.324,E2 -14859.324} C_VEL
LIN {X 0,Y 325.788,Z 384.842,A -85,B 0,C 180,E1 -14861.195,E2 -14861.195} C_VEL
LIN {X 0,Y 326.68,Z 377.721,A -85,B 0,C 180,E1 -14863.372,E2 -14863.372} C_VEL
LIN {X 0,Y 327.806,Z 368.892,A -85,B 0,C 180,E1 -14865.544,E2 -14865.544} C_VEL
LIN {X 0,Y 329.138,Z 359.642,A -85,B 0,C 180,E1 -14867.394,E2 -14867.394} C_VEL
LIN {X 0,Y 330.545,Z 349.416,A -85,B 0,C 180,E1 -14869.081,E2 -14869.081} C_VEL
LIN {X 0,Y 332.186,Z 338.179,A -85,B 0,C 180,E1 -14870.593,E2 -14870.593} C_VEL
LIN {X 0,Y 333.684,Z 326.536,A -85,B 0,C 180,E1 -14871.871,E2 -14871.871} C_VEL
LIN {X 0,Y 335.178,Z 313.752,A -85,B 0,C 180,E1 -14872.987,E2 -14872.987} C_VEL
LIN {X 0,Y 336.403,Z 300.613,A -85,B 0,C 180,E1 -14873.877,E2 -14873.877} C_VEL
LIN {X 0,Y 337.514,Z 286.472,A -85,B 0,C 180,E1 -14874.57,E2 -14874.57} C_VEL
LIN {X 0,Y 338.252,Z 271.536,A -85,B 0,C 180,E1 -14875.045,E2 -14875.045} C_VEL
LIN {X 0,Y 340.333,Z 179.853,A -85,B 0,C 180,E1 -14876.977,E2 -14876.977} C_VEL
LIN {X 0,Y 334.978,Z 147.816,A -85,B 0,C 180,E1 -14878.137,E2 -14878.137} C_VEL
LIN {X 0,Y 331.157,Z 138.022,A -85,B 0,C 180,E1 -14878.718,E2 -14878.718} C_VEL
LIN {X 0,Y 328.489,Z 125.651,A -85,B 0,C 180,E1 -14882.039,E2 -14882.039} C_VEL
LIN {X 0,Y 326.62,Z 117.929,A -85,B 0,C 180,E1 -14884.25,E2 -14884.25} C_VEL
LIN {X 0,Y 326.627,Z 117.925,A -85,B 0,C 180,E1 -14887.238,E2 -14887.238} C_VEL
LIN {X 0,Y 326.577,Z 117.928,A -85,B 0,C 180,E1 -14891.131,E2 -14891.131} C_VEL
LIN {X 0,Y 326.585,Z 117.927,A -85,B 0,C 180,E1 -14894.753,E2 -14894.753} C_VEL
LIN {X 0,Y 326.622,Z 117.924,A -85,B 0,C 180,E1 -14898.162,E2 -14898.162} C_VEL
LIN {X 0,Y 326.642,Z 117.916,A -85,B 0,C 180,E1 -14901.394,E2 -14901.394} C_VEL
LIN {X 0,Y 326.618,Z 117.923,A -85,B 0,C 180,E1 -14904.851,E2 -14904.851} C_VEL
LIN {X 0,Y 326.606,Z 117.928,A -85,B 0,C 180,E1 -14907.455,E2 -14907.455} C_VEL
LIN {X 0,Y 326.659,Z 117.916,A -85,B 0,C 180,E1 -14910.341,E2 -14910.341} C_VEL
LIN {X 0,Y 326.689,Z 117.914,A -85,B 0,C 180,E1 -14914.516,E2 -14914.516} C_VEL
LIN {X 0,Y 326.647,Z 117.92,A -85,B 0,C 180,E1 -14918.546,E2 -14918.546} C_VEL
LIN {X 0,Y 326.743,Z 117.907,A -85,B 0,C 180,E1 -14921.178,E2 -14921.178} C_VEL
LIN {X 0,Y 326.762,Z 117.904,A -85,B 0,C 180,E1 -14925.433,E2 -14925.433} C_VEL
LIN {X 0,Y 326.769,Z 117.907,A -85,B 0,C 180,E1 -14928.839,E2 -14928.839} C_VEL
LIN {X 0,Y 326.957,Z 117.883,A -85,B 0,C 180,E1 -14932.59,E2 -14932.59} C_VEL
LIN {X 0,Y 326.774,Z 117.902,A -85,B 0,C 180,E1 -14935.065,E2 -14935.065} C_VEL
LIN {X 0,Y 327.045,Z 117.869,A -85,B 0,C 180,E1 -14937.537,E2 -14937.537} C_VEL
LIN {X 0,Y 327.196,Z 117.852,A -85,B 0,C 180,E1 -14940,E2 -14940} C_VEL
LIN {X 0,Y 327.045,Z 117.869,A -85,B 0,C 180,E1 -14942.463,E2 -14942.463} C_VEL
LIN {X 0,Y 326.931,Z 117.885,A -85,B 0,C 180,E1 -14946.499,E2 -14946.499} C_VEL
LIN {X 0,Y 326.804,Z 117.898,A -85,B 0,C 180,E1 -14949.907,E2 -14949.907} C_VEL
LIN {X 0,Y 326.758,Z 117.908,A -85,B 0,C 180,E1 -14953.686,E2 -14953.686} C_VEL
LIN {X 0,Y 326.699,Z 117.912,A -85,B 0,C 180,E1 -14957.528,E2 -14957.528} C_VEL
LIN {X 0,Y 326.665,Z 117.918,A -85,B 0,C 180,E1 -14960.135,E2 -14960.135} C_VEL
LIN {X 0,Y 326.652,Z 117.915,A -85,B 0,C 180,E1 -14964.129,E2 -14964.129} C_VEL
LIN {X 0,Y 326.682,Z 117.914,A -85,B 0,C 180,E1 -14966.858,E2 -14966.858} C_VEL
LIN {X 0,Y 326.634,Z 117.919,A -85,B 0,C 180,E1 -14970.61,E2 -14970.61} C_VEL
LIN {X 0,Y 326.607,Z 117.924,A -85,B 0,C 180,E1 -14974.02,E2 -14974.02} C_VEL
LIN {X 0,Y 326.627,Z 117.923,A -85,B 0,C 180,E1 -14977.239,E2 -14977.239} C_VEL
LIN {X 0,Y 326.578,Z 117.929,A -85,B 0,C 180,E1 -14981.132,E2 -14981.132} C_VEL
LIN {X 0,Y 326.557,Z 117.935,A -85,B 0,C 180,E1 -14984.748,E2 -14984.748} C_VEL
LIN {X 0,Y 326.576,Z 117.929,A -85,B 0,C 180,E1 -14988.155,E2 -14988.155} C_VEL
LIN {X 0,Y 326.598,Z 117.92,A -85,B 0,C 180,E1 -14991.388,E2 -14991.388} C_VEL
LIN {X 0,Y 326.621,Z 117.925,A -85,B 0,C 180,E1 -14994.852,E2 -14994.852} C_VEL
LIN {X 0,Y 326.609,Z 117.924,A -85,B 0,C 180,E1 -14997.456,E2 -14997.456} C_VEL
LIN {X 0,Y 326.618,Z 117.927,A -85,B 0,C 180,E1 -15000.337,E2 -15000.337} C_VEL
LIN {X 0,Y 326.643,Z 117.921,A -85,B 0,C 180,E1 -15004.645,E2 -15004.645} C_VEL
LIN {X 0,Y 326.664,Z 118.011,A -85,B 0,C 180,E1 -15004.99,E2 -15004.99} C_VEL
LIN {X 0,Y 328.323,Z 125.2,A -85,B 0,C 180,E1 -15007.14,E2 -15007.14} C_VEL
LIN {X 0,Y 337.612,Z 147.936,A -85,B 0,C 180,E1 -15008.453,E2 -15008.453} C_VEL
LIN {X 0,Y 339.821,Z 154.634,A -85,B 0,C 180,E1 -15008.783,E2 -15008.783} C_VEL
LIN {X 0,Y 340.864,Z 160.023,A -85,B 0,C 180,E1 -15008.987,E2 -15008.987} C_VEL
LIN {X 0,Y 338.392,Z 261.816,A -85,B 0,C 180,E1 -15011.143,E2 -15011.143} C_VEL
LIN {X 0,Y 337.71,Z 276.331,A -85,B 0,C 180,E1 -15011.693,E2 -15011.693} C_VEL
LIN {X 0,Y 336.651,Z 290.227,A -85,B 0,C 180,E1 -15012.459,E2 -15012.459} C_VEL
LIN {X 0,Y 335.41,Z 303.151,A -85,B 0,C 180,E1 -15013.412,E2 -15013.412} C_VEL
LIN {X 0,Y 333.962,Z 315.678,A -85,B 0,C 180,E1 -15014.593,E2 -15014.593} C_VEL
LIN {X 0,Y 332.502,Z 327.095,A -85,B 0,C 180,E1 -15015.932,E2 -15015.932} C_VEL
LIN {X 0,Y 330.96,Z 337.589,A -85,B 0,C 180,E1 -15017.429,E2 -15017.429} C_VEL
LIN {X 0,Y 329.593,Z 347.991,A -85,B 0,C 180,E1 -15019.247,E2 -15019.247} C_VEL
LIN {X 0,Y 328.301,Z 356.595,A -85,B 0,C 180,E1 -15021.072,E2 -15021.072} C_VEL
LIN {X 0,Y 327.109,Z 364.859,A -85,B 0,C 180,E1 -15023.214,E2 -15023.214} C_VEL
LIN {X 0,Y 326.18,Z 370.624,A -85,B 0,C 180,E1 -15025.056,E2 -15025.056} C_VEL
LIN {X 0,Y 325.524,Z 376.786,A -85,B 0,C 180,E1 -15027.525,E2 -15027.525} C_VEL
LIN {X 0,Y 325.085,Z 381.317,A -85,B 0,C 180,E1 -15030,E2 -15030} C_VEL
LIN {X 0,Y 324.873,Z 384.397,A -85,B 0,C 180,E1 -15032.48,E2 -15032.48} C_VEL
LIN {X 0,Y 324.866,Z 386.12,A -85,B 0,C 180,E1 -15034.964,E2 -15034.964} C_VEL
LIN {X 0,Y 324.884,Z 386.486,A -85,B 0,C 180,E1 -15036.21,E2 -15036.21} C_VEL
LIN {X 0,Y 324.811,Z 386.231,A -85,B 0,C 180,E1 -15038.712,E2 -15038.712} C_VEL
LIN {X 0,Y 325.008,Z 384.635,A -85,B 0,C 180,E1 -15041.223,E2 -15041.223} C_VEL
LIN {X 0,Y 325.574,Z 381.658,A -85,B 0,C 180,E1 -15043.736,E2 -15043.736} C_VEL
LIN {X 0,Y 326.268,Z 377.209,A -85,B 0,C 180,E1 -15046.262,E2 -15046.262} C_VEL
LIN {X 0,Y 327.113,Z 372.763,A -85,B 0,C 180,E1 -15048.152,E2 -15048.152} C_VEL
LIN {X 0,Y 328.423,Z 366.309,A -85,B 0,C 180,E1 -15050.349,E2 -15050.349} C_VEL
LIN {X 0,Y 330.006,Z 358.255,A -85,B 0,C 180,E1 -15052.541,E2 -15052.541} C_VEL
LIN {X 0,Y 331.956,Z 348.908,A -85,B 0,C 180,E1 -15054.576,E2 -15054.576} C_VEL
LIN {X 0,Y 333.705,Z 339.55,A -85,B 0,C 180,E1 -15056.249,E2 -15056.249} C_VEL
LIN {X 0,Y 335.644,Z 329.197,A -85,B 0,C 180,E1 -15057.768,E2 -15057.768} C_VEL
LIN {X 0,Y 337.746,Z 316.739,A -85,B 0,C 180,E1 -15059.245,E2 -15059.245} C_VEL
LIN {X 0,Y 339.367,Z 305.594,A -85,B 0,C 180,E1 -15060.317,E2 -15060.317} C_VEL
LIN {X 0,Y 340.974,Z 292.993,A -85,B 0,C 180,E1 -15061.276,E2 -15061.276} C_VEL
LIN {X 0,Y 342.269,Z 278.838,A -85,B 0,C 180,E1 -15062.094,E2 -15062.094} C_VEL
LIN {X 0,Y 343.315,Z 264.37,A -85,B 0,C 180,E1 -15062.66,E2 -15062.66} C_VEL
LIN {X 0,Y 343.968,Z 245.558,A -85,B 0,C 180,E1 -15063.106,E2 -15063.106} C_VEL
LIN {X 0,Y 343.596,Z 239.757,A -85,B 0,C 180,E1 -15063.278,E2 -15063.278} C_VEL
LIN {X 0,Y 339.231,Z 221.119,A -85,B 0,C 180,E1 -15064.151,E2 -15064.151} C_VEL
LIN {X 0,Y 338.825,Z 215.319,A -85,B 0,C 180,E1 -15064.332,E2 -15064.332} C_VEL
LIN {X 0,Y 340.241,Z 165.041,A -85,B 0,C 180,E1 -15065.409,E2 -15065.409} C_VEL
LIN {X 0,Y 333.275,Z 149.183,A -85,B 0,C 180,E1 -15066.56,E2 -15066.56} C_VEL
LIN {X 0,Y 325.474,Z 133.38,A -85,B 0,C 180,E1 -15067.876,E2 -15067.876} C_VEL
LIN {X 0,Y 321.364,Z 125.677,A -85,B 0,C 180,E1 -15068.612,E2 -15068.612} C_VEL
LIN {X 0,Y 319.516,Z 118.81,A -85,B 0,C 180,E1 -15071.078,E2 -15071.078} C_VEL
LIN {X 0,Y 319.519,Z 118.81,A -85,B 0,C 180,E1 -15073.46,E2 -15073.46} C_VEL
LIN {X 0,Y 319.552,Z 118.801,A -85,B 0,C 180,E1 -15077.016,E2 -15077.016} C_VEL
LIN {X 0,Y 319.515,Z 118.79,A -85,B 0,C 180,E1 -15080.366,E2 -15080.366} C_VEL
LIN {X 0,Y 319.579,Z 118.797,A -85,B 0,C 180,E1 -15084.457,E2 -15084.457} C_VEL
LIN {X 0,Y 319.525,Z 118.808,A -85,B 0,C 180,E1 -15088.137,E2 -15088.137} C_VEL
LIN {X 0,Y 319.572,Z 118.803,A -85,B 0,C 180,E1 -15091.603,E2 -15091.603} C_VEL
LIN {X 0,Y 319.574,Z 118.804,A -85,B 0,C 180,E1 -15095.301,E2 -15095.301} C_VEL
LIN {X 0,Y 319.567,Z 118.794,A -85,B 0,C 180,E1 -15098.045,E2 -15098.045} C_VEL
LIN {X 0,Y 319.659,Z 118.785,A -85,B 0,C 180,E1 -15100.979,E2 -15100.979} C_VEL
LIN {X 0,Y 319.713,Z 118.78,A -85,B 0,C 180,E1 -15105.289,E2 -15105.289} C_VEL
LIN {X 0,Y 319.724,Z 118.786,A -85,B 0,C 180,E1 -15108.589,E2 -15108.589} C_VEL
LIN {X 0,Y 319.859,Z 118.762,A -85,B 0,C 180,E1 -15112.424,E2 -15112.424} C_VEL
LIN {X 0,Y 319.734,Z 118.777,A -85,B 0,C 180,E1 -15114.956,E2 -15114.956} C_VEL
LIN {X 0,Y 319.986,Z 118.745,A -85,B 0,C 180,E1 -15117.482,E2 -15117.482} C_VEL
LIN {X 0,Y 320.131,Z 118.727,A -85,B 0,C 180,E1 -15120,E2 -15120} C_VEL
LIN {X 0,Y 319.986,Z 118.747,A -85,B 0,C 180,E1 -15122.517,E2 -15122.517} C_VEL
LIN {X 0,Y 319.902,Z 118.749,A -85,B 0,C 180,E1 -15126.306,E2 -15126.306} C_VEL
LIN {X 0,Y 319.736,Z 118.777,A -85,B 0,C 180,E1 -15130.128,E2 -15130.128} C_VEL
LIN {X 0,Y 319.733,Z 118.782,A -85,B 0,C 180,E1 -15133.992,E2 -15133.992} C_VEL
LIN {X 0,Y 319.659,Z 118.79,A -85,B 0,C 180,E1 -15137.927,E2 -15137.927} C_VEL
LIN {X 0,Y 319.614,Z 118.786,A -85,B 0,C 180,E1 -15140.599,E2 -15140.599} C_VEL
LIN {X 0,Y 319.571,Z 118.8,A -85,B 0,C 180,E1 -15143.319,E2 -15143.319} C_VEL
LIN {X 0,Y 319.635,Z 118.79,A -85,B 0,C 180,E1 -15146.088,E2 -15146.088} C_VEL
LIN {X 0,Y 319.59,Z 118.793,A -85,B 0,C 180,E1 -15148.933,E2 -15148.933} C_VEL
LIN {X 0,Y 319.533,Z 118.803,A -85,B 0,C 180,E1 -15151.862,E2 -15151.862} C_VEL
LIN {X 0,Y 319.58,Z 118.795,A -85,B 0,C 180,E1 -15155.543,E2 -15155.543} C_VEL
LIN {X 0,Y 319.559,Z 118.783,A -85,B 0,C 180,E1 -15159.669,E2 -15159.669} C_VEL
LIN {X 0,Y 319.522,Z 118.8,A -85,B 0,C 180,E1 -15163.46,E2 -15163.46} C_VEL
LIN {X 0,Y 319.554,Z 118.805,A -85,B 0,C 180,E1 -15167.016,E2 -15167.016} C_VEL
LIN {X 0,Y 319.596,Z 118.795,A -85,B 0,C 180,E1 -15171.191,E2 -15171.191} C_VEL
LIN {X 0,Y 319.617,Z 118.969,A -85,B 0,C 180,E1 -15171.898,E2 -15171.898} C_VEL
LIN {X 0,Y 322.325,Z 128.698,A -85,B 0,C 180,E1 -15175.101,E2 -15175.101} C_VEL
LIN {X 0,Y 324.566,Z 137.807,A -85,B 0,C 180,E1 -15177.858,E2 -15177.858} C_VEL
LIN {X 0,Y 334.217,Z 158.258,A -85,B 0,C 180,E1 -15179.502,E2 -15179.502} C_VEL
LIN {X 0,Y 335.641,Z 162.063,A -85,B 0,C 180,E1 -15179.753,E2 -15179.753} C_VEL
LIN {X 0,Y 339.714,Z 183.506,A -85,B 0,C 180,E1 -15180.714,E2 -15180.714} C_VEL
LIN {X 0,Y 336.923,Z 276.409,A -85,B 0,C 180,E1 -15182.725,E2 -15182.725} C_VEL
LIN {X 0,Y 335.8,Z 290.762,A -85,B 0,C 180,E1 -15183.258,E2 -15183.258} C_VEL
LIN {X 0,Y 334.206,Z 305.135,A -85,B 0,C 180,E1 -15184.045,E2 -15184.045} C_VEL
LIN {X 0,Y 332.459,Z 317.889,A -85,B 0,C 180,E1 -15184.989,E2 -15184.989} C_VEL
LIN {X 0,Y 330.474,Z 331.221,A -85,B 0,C 180,E1 -15186.274,E2 -15186.274} C_VEL
LIN {X 0,Y 328.389,Z 342.851,A -85,B 0,C 180,E1 -15187.674,E2 -15187.674} C_VEL
LIN {X 0,Y 326.367,Z 353.117,A -85,B 0,C 180,E1 -15189.187,E2 -15189.187} C_VEL
LIN {X 0,Y 324.283,Z 363.354,A -85,B 0,C 180,E1 -15191.029,E2 -15191.029} C_VEL
LIN {X 0,Y 322.465,Z 371.836,A -85,B 0,C 180,E1 -15192.889,E2 -15192.889} C_VEL
LIN {X 0,Y 320.853,Z 379.957,A -85,B 0,C 180,E1 -15195.086,E2 -15195.086} C_VEL
LIN {X 0,Y 319.625,Z 386.522,A -85,B 0,C 180,E1 -15197.298,E2 -15197.298} C_VEL
LIN {X 0,Y 318.587,Z 392.365,A -85,B 0,C 180,E1 -15199.835,E2 -15199.835} C_VEL
LIN {X 0,Y 318.024,Z 396.655,A -85,B 0,C 180,E1 -15202.38,E2 -15202.38} C_VEL
LIN {X 0,Y 317.784,Z 399.517,A -85,B 0,C 180,E1 -15204.925,E2 -15204.925} C_VEL
LIN {X 0,Y 317.74,Z 401.024,A -85,B 0,C 180,E1 -15207.464,E2 -15207.464} C_VEL
LIN {X 0,Y 317.736,Z 401.2,A -85,B 0,C 180,E1 -15210,E2 -15210} C_VEL
LIN {X 0,Y 317.747,Z 400.042,A -85,B 0,C 180,E1 -15212.535,E2 -15212.535} C_VEL
LIN {X 0,Y 317.768,Z 397.519,A -85,B 0,C 180,E1 -15215.075,E2 -15215.075} C_VEL
LIN {X 0,Y 317.97,Z 393.53,A -85,B 0,C 180,E1 -15217.621,E2 -15217.621} C_VEL
LIN {X 0,Y 318.432,Z 387.955,A -85,B 0,C 180,E1 -15220.17,E2 -15220.17} C_VEL
LIN {X 0,Y 319.212,Z 381.655,A -85,B 0,C 180,E1 -15222.396,E2 -15222.396} C_VEL
LIN {X 0,Y 320.205,Z 374.072,A -85,B 0,C 180,E1 -15224.546,E2 -15224.546} C_VEL
LIN {X 0,Y 321.307,Z 365.563,A -85,B 0,C 180,E1 -15226.52,E2 -15226.52} C_VEL
LIN {X 0,Y 322.809,Z 355.647,A -85,B 0,C 180,E1 -15228.402,E2 -15228.402} C_VEL
LIN {X 0,Y 324.486,Z 344.622,A -85,B 0,C 180,E1 -15230.11,E2 -15230.11} C_VEL
LIN {X 0,Y 326.257,Z 332.624,A -85,B 0,C 180,E1 -15231.616,E2 -15231.616} C_VEL
LIN {X 0,Y 327.77,Z 320.203,A -85,B 0,C 180,E1 -15232.869,E2 -15232.869} C_VEL
LIN {X 0,Y 329.205,Z 306.694,A -85,B 0,C 180,E1 -15233.93,E2 -15233.93} C_VEL
LIN {X 0,Y 330.532,Z 292.604,A -85,B 0,C 180,E1 -15234.747,E2 -15234.747} C_VEL
LIN {X 0,Y 331.467,Z 277.715,A -85,B 0,C 180,E1 -15235.342,E2 -15235.342} C_VEL
LIN {X 0,Y 332.277,Z 251.31,A -85,B 0,C 180,E1 -15235.948,E2 -15235.948} C_VEL
LIN {X 0,Y 333.895,Z 180.955,A -85,B 0,C 180,E1 -15237.453,E2 -15237.453} C_VEL
LIN {X 0,Y 328.867,Z 150.477,A -85,B 0,C 180,E1 -15238.584,E2 -15238.584} C_VEL
LIN {X 0,Y 323.933,Z 137.924,A -85,B 0,C 180,E1 -15239.33,E2 -15239.33} C_VEL
LIN {X 0,Y 321.217,Z 125.445,A -85,B 0,C 180,E1 -15242.786,E2 -15242.786} C_VEL
LIN {X 0,Y 319.617,Z 118.801,A -85,B 0,C 180,E1 -15244.779,E2 -15244.779} C_VEL
LIN {X 0,Y 319.572,Z 118.806,A -85,B 0,C 180,E1 -15248.008,E2 -15248.008} C_VEL
LIN {X 0,Y 319.525,Z 118.809,A -85,B 0,C 180,E1 -15251.597,E2 -15251.597} C_VEL
LIN {X 0,Y 319.576,Z 118.801,A -85,B 0,C 180,E1 -15255.273,E2 -15255.273} C_VEL
LIN {X 0,Y 319.579,Z 118.799,A -85,B 0,C 180,E1 -15258.72,E2 -15258.72} C_VEL
LIN {X 0,Y 319.58,Z 118.796,A -85,B 0,C 180,E1 -15262.343,E2 -15262.343} C_VEL
LIN {X 0,Y 319.559,Z 118.804,A -85,B 0,C 180,E1 -15265.123,E2 -15265.123} C_VEL
LIN {X 0,Y 319.569,Z 118.804,A -85,B 0,C 180,E1 -15269.058,E2 -15269.058} C_VEL
LIN {X 0,Y 319.607,Z 118.796,A -85,B 0,C 180,E1 -15272.498,E2 -15272.498} C_VEL
LIN {X 0,Y 319.604,Z 118.797,A -85,B 0,C 180,E1 -15275.304,E2 -15275.304} C_VEL
LIN {X 0,Y 319.596,Z 118.797,A -85,B 0,C 180,E1 -15278.048,E2 -15278.048} C_VEL
LIN {X 0,Y 319.688,Z 118.786,A -85,B 0,C 180,E1 -15280.962,E2 -15280.962} C_VEL
LIN {X 0,Y 319.73,Z 118.781,A -85,B 0,C 180,E1 -15285.276,E2 -15285.276} C_VEL
LIN {X 0,Y 319.755,Z 118.777,A -85,B 0,C 180,E1 -15289.873,E2 -15289.873} C_VEL
LIN {X 0,Y 319.911,Z 118.762,A -85,B 0,C 180,E1 -15292.426,E2 -15292.426} C_VEL
LIN {X 0,Y 319.744,Z 118.778,A -85,B 0,C 180,E1 -15294.956,E2 -15294.956} C_VEL
LIN {X 0,Y 319.989,Z 118.748,A -85,B 0,C 180,E1 -15297.483,E2 -15297.483} C_VEL
LIN {X 0,Y 320.148,Z 118.73,A -85,B 0,C 180,E1 -15300,E2 -15300} C_VEL
LIN {X 0,Y 319.988,Z 118.747,A -85,B 0,C 180,E1 -15302.518,E2 -15302.518} C_VEL
LIN {X 0,Y 319.896,Z 118.761,A -85,B 0,C 180,E1 -15306.483,E2 -15306.483} C_VEL
LIN {X 0,Y 319.751,Z 118.776,A -85,B 0,C 180,E1 -15310.128,E2 -15310.128} C_VEL
LIN {X 0,Y 319.73,Z 118.78,A -85,B 0,C 180,E1 -15314.724,E2 -15314.724} C_VEL
LIN {X 0,Y 319.688,Z 118.783,A -85,B 0,C 180,E1 -15319.038,E2 -15319.038} C_VEL
LIN {X 0,Y 319.57,Z 118.803,A -85,B 0,C 180,E1 -15323.32,E2 -15323.32} C_VEL
LIN {X 0,Y 319.634,Z 118.791,A -85,B 0,C 180,E1 -15326.088,E2 -15326.088} C_VEL
LIN {X 0,Y 319.58,Z 118.801,A -85,B 0,C 180,E1 -15328.935,E2 -15328.935} C_VEL
LIN {X 0,Y 319.53,Z 118.804,A -85,B 0,C 180,E1 -15331.862,E2 -15331.862} C_VEL
LIN {X 0,Y 319.58,Z 118.8,A -85,B 0,C 180,E1 -15335.543,E2 -15335.543} C_VEL
LIN {X 0,Y 319.559,Z 118.803,A -85,B 0,C 180,E1 -15339.669,E2 -15339.669} C_VEL
LIN {X 0,Y 319.558,Z 118.803,A -85,B 0,C 180,E1 -15343.468,E2 -15343.468} C_VEL
LIN {X 0,Y 319.56,Z 118.805,A -85,B 0,C 180,E1 -15347.018,E2 -15347.018} C_VEL
LIN {X 0,Y 319.547,Z 118.801,A -85,B 0,C 180,E1 -15350.371,E2 -15350.371} C_VEL
LIN {X 0,Y 319.581,Z 118.804,A -85,B 0,C 180,E1 -15354.457,E2 -15354.457} C_VEL
LIN {X 0,Y 319.525,Z 118.809,A -85,B 0,C 180,E1 -15358.138,E2 -15358.138} C_VEL
LIN {X 0,Y 319.573,Z 118.802,A -85,B 0,C 180,E1 -15361.604,E2 -15361.604} C_VEL
LIN {X 0,Y 319.614,Z 118.891,A -85,B 0,C 180,E1 -15364.504,E2 -15364.504} C_VEL
LIN {X 0,Y 321.124,Z 125.295,A -85,B 0,C 180,E1 -15366.478,E2 -15366.478} C_VEL
LIN {X 0,Y 330.102,Z 146.801,A -85,B 0,C 180,E1 -15367.808,E2 -15367.808} C_VEL
LIN {X 0,Y 333.59,Z 156.769,A -85,B 0,C 180,E1 -15368.333,E2 -15368.333} C_VEL
LIN {X 0,Y 334.389,Z 162.128,A -85,B 0,C 180,E1 -15368.523,E2 -15368.523} C_VEL
LIN {X 0,Y 331.856,Z 262.03,A -85,B 0,C 180,E1 -15370.677,E2 -15370.677} C_VEL
LIN {X 0,Y 331.153,Z 276.525,A -85,B 0,C 180,E1 -15371.237,E2 -15371.237} C_VEL
LIN {X 0,Y 330.184,Z 289.287,A -85,B 0,C 180,E1 -15371.943,E2 -15371.943} C_VEL
LIN {X 0,Y 328.862,Z 302.457,A -85,B 0,C 180,E1 -15372.912,E2 -15372.912} C_VEL
LIN {X 0,Y 327.525,Z 313.738,A -85,B 0,C 180,E1 -15373.963,E2 -15373.963} C_VEL
LIN {X 0,Y 325.993,Z 325.527,A -85,B 0,C 180,E1 -15375.326,E2 -15375.326} C_VEL
LIN {X 0,Y 324.381,Z 336.312,A -85,B 0,C 180,E1 -15376.851,E2 -15376.851} C_VEL
LIN {X 0,Y 322.945,Z 345.946,A -85,B 0,C 180,E1 -15378.504,E2 -15378.504} C_VEL
LIN {X 0,Y 321.676,Z 354.422,A -85,B 0,C 180,E1 -15380.252,E2 -15380.252} C_VEL
LIN {X 0,Y 320.533,Z 361.992,A -85,B 0,C 180,E1 -15382.124,E2 -15382.124} C_VEL
LIN {X 0,Y 319.483,Z 369.218,A -85,B 0,C 180,E1 -15384.319,E2 -15384.319} C_VEL
LIN {X 0,Y 318.635,Z 375.718,A -85,B 0,C 180,E1 -15386.839,E2 -15386.839} C_VEL
LIN {X 0,Y 318.142,Z 380.6,A -85,B 0,C 180,E1 -15389.367,E2 -15389.367} C_VEL
LIN {X 0,Y 317.827,Z 383.288,A -85,B 0,C 180,E1 -15391.267,E2 -15391.267} C_VEL
LIN {X 0,Y 317.802,Z 385.638,A -85,B 0,C 180,E1 -15393.804,E2 -15393.804} C_VEL
LIN {X 0,Y 317.792,Z 386.66,A -85,B 0,C 180,E1 -15396.349,E2 -15396.349} C_VEL
LIN {X 0,Y 317.73,Z 386.364,A -85,B 0,C 180,E1 -15398.907,E2 -15398.907} C_VEL
LIN {X 0,Y 317.957,Z 384.727,A -85,B 0,C 180,E1 -15401.475,E2 -15401.475} C_VEL
LIN {X 0,Y 318.551,Z 381.706,A -85,B 0,C 180,E1 -15404.045,E2 -15404.045} C_VEL
LIN {X 0,Y 319.315,Z 377.21,A -85,B 0,C 180,E1 -15406.626,E2 -15406.626} C_VEL
LIN {X 0,Y 320.242,Z 372.717,A -85,B 0,C 180,E1 -15408.555,E2 -15408.555} C_VEL
LIN {X 0,Y 321.608,Z 366.21,A -85,B 0,C 180,E1 -15410.8,E2 -15410.8} C_VEL
LIN {X 0,Y 323.327,Z 358.1,A -85,B 0,C 180,E1 -15413.033,E2 -15413.033} C_VEL
LIN {X 0,Y 325.3,Z 349.068,A -85,B 0,C 180,E1 -15415.027,E2 -15415.027} C_VEL
LIN {X 0,Y 327.212,Z 339.211,A -85,B 0,C 180,E1 -15416.811,E2 -15416.811} C_VEL
LIN {X 0,Y 329.263,Z 328.756,A -85,B 0,C 180,E1 -15418.354,E2 -15418.354} C_VEL
LIN {X 0,Y 331.267,Z 317.359,A -85,B 0,C 180,E1 -15419.729,E2 -15419.729} C_VEL
LIN {X 0,Y 332.904,Z 306.625,A -85,B 0,C 180,E1 -15420.794,E2 -15420.794} C_VEL
LIN {X 0,Y 334.705,Z 293.136,A -85,B 0,C 180,E1 -15421.841,E2 -15421.841} C_VEL
LIN {X 0,Y 336.055,Z 278.977,A -85,B 0,C 180,E1 -15422.672,E2 -15422.672} C_VEL
LIN {X 0,Y 337.165,Z 264.02,A -85,B 0,C 180,E1 -15423.262,E2 -15423.262} C_VEL
LIN {X 0,Y 338.05,Z 238.03,A -85,B 0,C 180,E1 -15423.861,E2 -15423.861} C_VEL
LIN {X 0,Y 338.825,Z 215.319,A -85,B 0,C 180,E1 -15424.332,E2 -15424.332} C_VEL
LIN {X 0,Y 338.416,Z 209.522,A -85,B 0,C 180,E1 -15424.515,E2 -15424.515} C_VEL
LIN {X 0,Y 334.064,Z 190.918,A -85,B 0,C 180,E1 -15425.427,E2 -15425.427} C_VEL
LIN {X 0,Y 333.685,Z 185.121,A -85,B 0,C 180,E1 -15425.613,E2 -15425.613} C_VEL
LIN {X 0,Y 334.128,Z 166.859,A -85,B 0,C 180,E1 -15426.021,E2 -15426.021} C_VEL
LIN {X 0,Y 326.696,Z 150.042,A -85,B 0,C 180,E1 -15427.295,E2 -15427.295} C_VEL
LIN {X 0,Y 318.563,Z 134.028,A -85,B 0,C 180,E1 -15428.718,E2 -15428.718} C_VEL
LIN {X 0,Y 314.154,Z 125.866,A -85,B 0,C 180,E1 -15429.546,E2 -15429.546} C_VEL
LIN {X 0,Y 312.474,Z 119.687,A -85,B 0,C 180,E1 -15431.826,E2 -15431.826} C_VEL
LIN {X 0,Y 312.451,Z 119.676,A -85,B 0,C 180,E1 -15435.79,E2 -15435.79} C_VEL
LIN {X 0,Y 312.442,Z 119.675,A -85,B 0,C 180,E1 -15439.283,E2 -15439.283} C_VEL
LIN {X 0,Y 312.511,Z 119.683,A -85,B 0,C 180,E1 -15442.612,E2 -15442.612} C_VEL
LIN {X 0,Y 312.521,Z 119.679,A -85,B 0,C 180,E1 -15446.311,E2 -15446.311} C_VEL
LIN {X 0,Y 312.497,Z 119.677,A -85,B 0,C 180,E1 -15450.345,E2 -15450.345} C_VEL
LIN {X 0,Y 312.531,Z 119.672,A -85,B 0,C 180,E1 -15454.092,E2 -15454.092} C_VEL
LIN {X 0,Y 312.541,Z 119.668,A -85,B 0,C 180,E1 -15457.525,E2 -15457.525} C_VEL
LIN {X 0,Y 312.59,Z 119.662,A -85,B 0,C 180,E1 -15461.653,E2 -15461.653} C_VEL
LIN {X 0,Y 312.687,Z 119.653,A -85,B 0,C 180,E1 -15465.686,E2 -15465.686} C_VEL
LIN {X 0,Y 312.699,Z 119.658,A -85,B 0,C 180,E1 -15469.641,E2 -15469.641} C_VEL
LIN {X 0,Y 312.801,Z 119.638,A -85,B 0,C 180,E1 -15472.252,E2 -15472.252} C_VEL
LIN {X 0,Y 312.704,Z 119.653,A -85,B 0,C 180,E1 -15474.842,E2 -15474.842} C_VEL
LIN {X 0,Y 312.987,Z 119.622,A -85,B 0,C 180,E1 -15478.713,E2 -15478.713} C_VEL
LIN {X 0,Y 312.987,Z 119.61,A -85,B 0,C 180,E1 -15481.286,E2 -15481.286} C_VEL
LIN {X 0,Y 312.699,Z 119.655,A -85,B 0,C 180,E1 -15485.158,E2 -15485.158} C_VEL
LIN {X 0,Y 312.797,Z 119.641,A -85,B 0,C 180,E1 -15487.747,E2 -15487.747} C_VEL
LIN {X 0,Y 312.664,Z 119.652,A -85,B 0,C 180,E1 -15491.671,E2 -15491.671} C_VEL
LIN {X 0,Y 312.701,Z 119.656,A -85,B 0,C 180,E1 -15494.887,E2 -15494.887} C_VEL
LIN {X 0,Y 312.631,Z 119.664,A -85,B 0,C 180,E1 -15499.236,E2 -15499.236} C_VEL
LIN {X 0,Y 312.547,Z 119.675,A -85,B 0,C 180,E1 -15502.789,E2 -15502.789} C_VEL
LIN {X 0,Y 312.603,Z 119.665,A -85,B 0,C 180,E1 -15505.935,E2 -15505.935} C_VEL
LIN {X 0,Y 312.546,Z 119.674,A -85,B 0,C 180,E1 -15509.65,E2 -15509.65} C_VEL
LIN {X 0,Y 312.52,Z 119.681,A -85,B 0,C 180,E1 -15513.689,E2 -15513.689} C_VEL
LIN {X 0,Y 312.521,Z 119.681,A -85,B 0,C 180,E1 -15517.386,E2 -15517.386} C_VEL
LIN {X 0,Y 312.49,Z 119.667,A -85,B 0,C 180,E1 -15520.709,E2 -15520.709} C_VEL
LIN {X 0,Y 312.452,Z 119.674,A -85,B 0,C 180,E1 -15524.209,E2 -15524.209} C_VEL
LIN {X 0,Y 312.514,Z 119.681,A -85,B 0,C 180,E1 -15527.913,E2 -15527.913} C_VEL
LIN {X 0,Y 312.578,Z 119.843,A -85,B 0,C 180,E1 -15531.112,E2 -15531.112} C_VEL
LIN {X 0,Y 315.413,Z 130.085,A -85,B 0,C 180,E1 -15534.596,E2 -15534.596} C_VEL
LIN {X 0,Y 317.258,Z 137.579,A -85,B 0,C 180,E1 -15536.939,E2 -15536.939} C_VEL
LIN {X 0,Y 326.918,Z 157.44,A -85,B 0,C 180,E1 -15538.651,E2 -15538.651} C_VEL
LIN {X 0,Y 329.999,Z 164.883,A -85,B 0,C 180,E1 -15539.197,E2 -15539.197} C_VEL
LIN {X 0,Y 333.651,Z 184.575,A -85,B 0,C 180,E1 -15540.098,E2 -15540.098} C_VEL
LIN {X 0,Y 330.824,Z 275.543,A -85,B 0,C 180,E1 -15542.093,E2 -15542.093} C_VEL
LIN {X 0,Y 329.646,Z 290.134,A -85,B 0,C 180,E1 -15542.631,E2 -15542.631} C_VEL
LIN {X 0,Y 328.015,Z 304.624,A -85,B 0,C 180,E1 -15543.432,E2 -15543.432} C_VEL
LIN {X 0,Y 326.074,Z 318.332,A -85,B 0,C 180,E1 -15544.464,E2 -15544.464} C_VEL
LIN {X 0,Y 324.138,Z 330.639,A -85,B 0,C 180,E1 -15545.672,E2 -15545.672} C_VEL
LIN {X 0,Y 321.836,Z 343.085,A -85,B 0,C 180,E1 -15547.194,E2 -15547.194} C_VEL
LIN {X 0,Y 319.731,Z 353.287,A -85,B 0,C 180,E1 -15548.735,E2 -15548.735} C_VEL
LIN {X 0,Y 317.534,Z 363.449,A -85,B 0,C 180,E1 -15550.61,E2 -15550.61} C_VEL
LIN {X 0,Y 315.642,Z 371.889,A -85,B 0,C 180,E1 -15552.507,E2 -15552.507} C_VEL
LIN {X 0,Y 313.964,Z 379.965,A -85,B 0,C 180,E1 -15554.75,E2 -15554.75} C_VEL
LIN {X 0,Y 312.657,Z 386.496,A -85,B 0,C 180,E1 -15557.01,E2 -15557.01} C_VEL
LIN {X 0,Y 311.565,Z 392.307,A -85,B 0,C 180,E1 -15559.603,E2 -15559.603} C_VEL
LIN {X 0,Y 310.972,Z 396.566,A -85,B 0,C 180,E1 -15562.206,E2 -15562.206} C_VEL
LIN {X 0,Y 310.69,Z 399.4,A -85,B 0,C 180,E1 -15564.808,E2 -15564.808} C_VEL
LIN {X 0,Y 310.662,Z 400.881,A -85,B 0,C 180,E1 -15567.407,E2 -15567.407} C_VEL
LIN {X 0,Y 310.648,Z 401.03,A -85,B 0,C 180,E1 -15570,E2 -15570} C_VEL
LIN {X 0,Y 310.669,Z 399.846,A -85,B 0,C 180,E1 -15572.593,E2 -15572.593} C_VEL
LIN {X 0,Y 310.683,Z 397.289,A -85,B 0,C 180,E1 -15575.191,E2 -15575.191} C_VEL
LIN {X 0,Y 310.903,Z 393.262,A -85,B 0,C 180,E1 -15577.795,E2 -15577.795} C_VEL
LIN {X 0,Y 311.389,Z 387.653,A -85,B 0,C 180,E1 -15580.402,E2 -15580.402} C_VEL
LIN {X 0,Y 312.212,Z 381.318,A -85,B 0,C 180,E1 -15582.678,E2 -15582.678} C_VEL
LIN {X 0,Y 313.238,Z 373.779,A -85,B 0,C 180,E1 -15584.855,E2 -15584.855} C_VEL
LIN {X 0,Y 314.443,Z 365.143,A -85,B 0,C 180,E1 -15586.891,E2 -15586.891} C_VEL
LIN {X 0,Y 315.997,Z 355.175,A -85,B 0,C 180,E1 -15588.813,E2 -15588.813} C_VEL
LIN {X 0,Y 317.792,Z 344.092,A -85,B 0,C 180,E1 -15590.553,E2 -15590.553} C_VEL
LIN {X 0,Y 319.444,Z 333.075,A -85,B 0,C 180,E1 -15591.963,E2 -15591.963} C_VEL
LIN {X 0,Y 320.988,Z 321.133,A -85,B 0,C 180,E1 -15593.21,E2 -15593.21} C_VEL
LIN {X 0,Y 322.458,Z 308.015,A -85,B 0,C 180,E1 -15594.291,E2 -15594.291} C_VEL
LIN {X 0,Y 323.856,Z 293.686,A -85,B 0,C 180,E1 -15595.163,E2 -15595.163} C_VEL
LIN {X 0,Y 324.79,Z 280.566,A -85,B 0,C 180,E1 -15595.729,E2 -15595.729} C_VEL
LIN {X 0,Y 325.411,Z 264.906,A -85,B 0,C 180,E1 -15596.149,E2 -15596.149} C_VEL
LIN {X 0,Y 327.464,Z 182.007,A -85,B 0,C 180,E1 -15597.951,E2 -15597.951} C_VEL
LIN {X 0,Y 322.806,Z 153.226,A -85,B 0,C 180,E1 -15599.042,E2 -15599.042} C_VEL
LIN {X 0,Y 316.649,Z 137.694,A -85,B 0,C 180,E1 -15600.011,E2 -15600.011} C_VEL
LIN {X 0,Y 314.179,Z 126.401,A -85,B 0,C 180,E1 -15603.233,E2 -15603.233} C_VEL
LIN {X 0,Y 312.546,Z 119.681,A -85,B 0,C 180,E1 -15605.283,E2 -15605.283} C_VEL
LIN {X 0,Y 312.507,Z 119.683,A -85,B 0,C 180,E1 -15609.027,E2 -15609.027} C_VEL
LIN {X 0,Y 312.494,Z 119.684,A -85,B 0,C 180,E1 -15612.43,E2 -15612.43} C_VEL
LIN {X 0,Y 312.537,Z 119.679,A -85,B 0,C 180,E1 -15616.02,E2 -15616.02} C_VEL
LIN {X 0,Y 312.529,Z 119.674,A -85,B 0,C 180,E1 -15619.869,E2 -15619.869} C_VEL
LIN {X 0,Y 312.538,Z 119.672,A -85,B 0,C 180,E1 -15622.617,E2 -15622.617} C_VEL
LIN {X 0,Y 312.518,Z 119.676,A -85,B 0,C 180,E1 -15626.311,E2 -15626.311} C_VEL
LIN {X 0,Y 312.544,Z 119.674,A -85,B 0,C 180,E1 -15630.35,E2 -15630.35} C_VEL
LIN {X 0,Y 312.601,Z 119.668,A -85,B 0,C 180,E1 -15634.064,E2 -15634.064} C_VEL
LIN {X 0,Y 312.586,Z 119.672,A -85,B 0,C 180,E1 -15637.529,E2 -15637.529} C_VEL
LIN {X 0,Y 312.637,Z 119.661,A -85,B 0,C 180,E1 -15641.656,E2 -15641.656} C_VEL
LIN {X 0,Y 312.692,Z 119.656,A -85,B 0,C 180,E1 -15645.686,E2 -15645.686} C_VEL
LIN {X 0,Y 312.7,Z 119.656,A -85,B 0,C 180,E1 -15649.642,E2 -15649.642} C_VEL
LIN {X 0,Y 312.852,Z 119.64,A -85,B 0,C 180,E1 -15652.254,E2 -15652.254} C_VEL
LIN {X 0,Y 312.714,Z 119.654,A -85,B 0,C 180,E1 -15654.843,E2 -15654.843} C_VEL
LIN {X 0,Y 312.987,Z 119.622,A -85,B 0,C 180,E1 -15658.714,E2 -15658.714} C_VEL
LIN {X 0,Y 312.988,Z 119.615,A -85,B 0,C 180,E1 -15661.287,E2 -15661.287} C_VEL
LIN {X 0,Y 312.707,Z 119.655,A -85,B 0,C 180,E1 -15665.158,E2 -15665.158} C_VEL
LIN {X 0,Y 312.817,Z 119.644,A -85,B 0,C 180,E1 -15667.747,E2 -15667.747} C_VEL
LIN {X 0,Y 312.669,Z 119.658,A -85,B 0,C 180,E1 -15671.672,E2 -15671.672} C_VEL
LIN {X 0,Y 312.699,Z 119.656,A -85,B 0,C 180,E1 -15674.888,E2 -15674.888} C_VEL
LIN {X 0,Y 312.63,Z 119.662,A -85,B 0,C 180,E1 -15679.237,E2 -15679.237} C_VEL
LIN {X 0,Y 312.546,Z 119.675,A -85,B 0,C 180,E1 -15682.79,E2 -15682.79} C_VEL
LIN {X 0,Y 312.602,Z 119.668,A -85,B 0,C 180,E1 -15685.936,E2 -15685.936} C_VEL
LIN {X 0,Y 312.538,Z 119.677,A -85,B 0,C 180,E1 -15689.651,E2 -15689.651} C_VEL
LIN {X 0,Y 312.519,Z 119.68,A -85,B 0,C 180,E1 -15693.689,E2 -15693.689} C_VEL
LIN {X 0,Y 312.52,Z 119.68,A -85,B 0,C 180,E1 -15697.386,E2 -15697.386} C_VEL
LIN {X 0,Y 312.49,Z 119.686,A -85,B 0,C 180,E1 -15700.71,E2 -15700.71} C_VEL
LIN {X 0,Y 312.473,Z 119.686,A -85,B 0,C 180,E1 -15704.206,E2 -15704.206} C_VEL
LIN {X 0,Y 312.486,Z 119.684,A -85,B 0,C 180,E1 -15707.919,E2 -15707.919} C_VEL
LIN {X 0,Y 312.499,Z 119.674,A -85,B 0,C 180,E1 -15710.972,E2 -15710.972} C_VEL
LIN {X 0,Y 312.533,Z 119.681,A -85,B 0,C 180,E1 -15714.221,E2 -15714.221} C_VEL
LIN {X 0,Y 312.502,Z 119.682,A -85,B 0,C 180,E1 -15717.334,E2 -15717.334} C_VEL
LIN {X 0,Y 312.508,Z 119.682,A -85,B 0,C 180,E1 -15721.292,E2 -15721.292} C_VEL
LIN {X 0,Y 312.551,Z 119.749,A -85,B 0,C 180,E1 -15723.987,E2 -15723.987} C_VEL
LIN {X 0,Y 313.988,Z 125.674,A -85,B 0,C 180,E1 -15725.835,E2 -15725.835} C_VEL
LIN {X 0,Y 322.199,Z 144.891,A -85,B 0,C 180,E1 -15727.076,E2 -15727.076} C_VEL
LIN {X 0,Y 327.321,Z 158.594,A -85,B 0,C 180,E1 -15727.853,E2 -15727.853} C_VEL
LIN {X 0,Y 327.961,Z 163.602,A -85,B 0,C 180,E1 -15728.027,E2 -15728.027} C_VEL
LIN {X 0,Y 325.34,Z 262.227,A -85,B 0,C 180,E1 -15730.192,E2 -15730.192} C_VEL
LIN {X 0,Y 324.613,Z 276.709,A -85,B 0,C 180,E1 -15730.762,E2 -15730.762} C_VEL
LIN {X 0,Y 323.61,Z 289.467,A -85,B 0,C 180,E1 -15731.481,E2 -15731.481} C_VEL
LIN {X 0,Y 322.355,Z 301.755,A -85,B 0,C 180,E1 -15732.392,E2 -15732.392} C_VEL
LIN {X 0,Y 320.951,Z 313.206,A -85,B 0,C 180,E1 -15733.461,E2 -15733.461} C_VEL
LIN {X 0,Y 319.323,Z 325.122,A -85,B 0,C 180,E1 -15734.85,E2 -15734.85} C_VEL
LIN {X 0,Y 317.862,Z 335.029,A -85,B 0,C 180,E1 -15736.25,E2 -15736.25} C_VEL
LIN {X 0,Y 316.359,Z 344.288,A -85,B 0,C 180,E1 -15737.817,E2 -15737.817} C_VEL
LIN {X 0,Y 314.925,Z 353.575,A -85,B 0,C 180,E1 -15739.716,E2 -15739.716} C_VEL
LIN {X 0,Y 313.683,Z 361.296,A -85,B 0,C 180,E1 -15741.626,E2 -15741.626} C_VEL
LIN {X 0,Y 312.644,Z 367.72,A -85,B 0,C 180,E1 -15743.547,E2 -15743.547} C_VEL
LIN {X 0,Y 311.955,Z 373.05,A -85,B 0,C 180,E1 -15745.478,E2 -15745.478} C_VEL
LIN {X 0,Y 311.275,Z 378.672,A -85,B 0,C 180,E1 -15748.059,E2 -15748.059} C_VEL
LIN {X 0,Y 310.885,Z 381.872,A -85,B 0,C 180,E1 -15750,E2 -15750} C_VEL
LIN {X 0,Y 310.712,Z 384.866,A -85,B 0,C 180,E1 -15752.593,E2 -15752.593} C_VEL
LIN {X 0,Y 310.69,Z 386.508,A -85,B 0,C 180,E1 -15755.192,E2 -15755.192} C_VEL
LIN {X 0,Y 310.624,Z 386.832,A -85,B 0,C 180,E1 -15757.802,E2 -15757.802} C_VEL
LIN {X 0,Y 310.693,Z 385.828,A -85,B 0,C 180,E1 -15760.426,E2 -15760.426} C_VEL
LIN {X 0,Y 311.211,Z 383.464,A -85,B 0,C 180,E1 -15763.052,E2 -15763.052} C_VEL
LIN {X 0,Y 311.914,Z 379.679,A -85,B 0,C 180,E1 -15765.687,E2 -15765.687} C_VEL
LIN {X 0,Y 312.706,Z 375.777,A -85,B 0,C 180,E1 -15767.663,E2 -15767.663} C_VEL
LIN {X 0,Y 313.922,Z 370.204,A -85,B 0,C 180,E1 -15769.9,E2 -15769.9} C_VEL
LIN {X 0,Y 315.565,Z 362.81,A -85,B 0,C 180,E1 -15772.248,E2 -15772.248} C_VEL
LIN {X 0,Y 317.35,Z 355.216,A -85,B 0,C 180,E1 -15774.186,E2 -15774.186} C_VEL
LIN {X 0,Y 319.309,Z 346.057,A -85,B 0,C 180,E1 -15776.117,E2 -15776.117} C_VEL
LIN {X 0,Y 321.564,Z 334.916,A -85,B 0,C 180,E1 -15778.028,E2 -15778.028} C_VEL
LIN {X 0,Y 323.711,Z 324.463,A -85,B 0,C 180,E1 -15779.464,E2 -15779.464} C_VEL
LIN {X 0,Y 325.639,Z 312.714,A -85,B 0,C 180,E1 -15780.8,E2 -15780.8} C_VEL
LIN {X 0,Y 327.767,Z 299.497,A -85,B 0,C 180,E1 -15781.962,E2 -15781.962} C_VEL
LIN {X 0,Y 329.122,Z 287.447,A -85,B 0,C 180,E1 -15782.81,E2 -15782.81} C_VEL
LIN {X 0,Y 330.379,Z 273.397,A -85,B 0,C 180,E1 -15783.533,E2 -15783.533} C_VEL
LIN {X 0,Y 331.27,Z 259.099,A -85,B 0,C 180,E1 -15784.014,E2 -15784.014} C_VEL
LIN {X 0,Y 333.685,Z 185.121,A -85,B 0,C 180,E1 -15785.613,E2 -15785.613} C_VEL
LIN {X 0,Y 333.151,Z 179.351,A -85,B 0,C 180,E1 -15785.815,E2 -15785.815} C_VEL
LIN {X 0,Y 331.518,Z 173.917,A -85,B 0,C 180,E1 -15786.131,E2 -15786.131} C_VEL
LIN {X 0,Y 330.035,Z 170.506,A -85,B 0,C 180,E1 -15786.384,E2 -15786.384} C_VEL
LIN {X 0,Y 323.013,Z 157.164,A -85,B 0,C 180,E1 -15787.548,E2 -15787.548} C_VEL
LIN {X 0,Y 315.261,Z 141.32,A -85,B 0,C 180,E1 -15788.945,E2 -15788.945} C_VEL
LIN {X 0,Y 308.254,Z 128.776,A -85,B 0,C 180,E1 -15790.241,E2 -15790.241} C_VEL
LIN {X 0,Y 306.924,Z 126.04,A -85,B 0,C 180,E1 -15790.543,E2 -15790.543} C_VEL
LIN {X 0,Y 305.433,Z 120.564,A -85,B 0,C 180,E1 -15792.672,E2 -15792.672} C_VEL
LIN {X 0,Y 305.422,Z 120.553,A -85,B 0,C 180,E1 -15796.344,E2 -15796.344} C_VEL
LIN {X 0,Y 305.411,Z 120.546,A -85,B 0,C 180,E1 -15799.884,E2 -15799.884} C_VEL
LIN {X 0,Y 305.463,Z 120.556,A -85,B 0,C 180,E1 -15803.637,E2 -15803.637} C_VEL
LIN {X 0,Y 305.466,Z 120.556,A -85,B 0,C 180,E1 -15806.483,E2 -15806.483} C_VEL
LIN {X 0,Y 305.432,Z 120.558,A -85,B 0,C 180,E1 -15809.587,E2 -15809.587} C_VEL
LIN {X 0,Y 305.458,Z 120.56,A -85,B 0,C 180,E1 -15812.602,E2 -15812.602} C_VEL
LIN {X 0,Y 305.475,Z 120.559,A -85,B 0,C 180,E1 -15815.536,E2 -15815.536} C_VEL
LIN {X 0,Y 305.501,Z 120.555,A -85,B 0,C 180,E1 -15819.813,E2 -15819.813} C_VEL
LIN {X 0,Y 305.545,Z 120.542,A -85,B 0,C 180,E1 -15822.601,E2 -15822.601} C_VEL
LIN {X 0,Y 305.628,Z 120.534,A -85,B 0,C 180,E1 -15825.348,E2 -15825.348} C_VEL
LIN {X 0,Y 305.636,Z 120.537,A -85,B 0,C 180,E1 -15829.399,E2 -15829.399} C_VEL
LIN {X 0,Y 305.751,Z 120.514,A -85,B 0,C 180,E1 -15832.072,E2 -15832.072} C_VEL
LIN {X 0,Y 305.672,Z 120.53,A -85,B 0,C 180,E1 -15834.723,E2 -15834.723} C_VEL
LIN {X 0,Y 305.954,Z 120.499,A -85,B 0,C 180,E1 -15838.684,E2 -15838.684} C_VEL
LIN {X 0,Y 305.954,Z 120.486,A -85,B 0,C 180,E1 -15841.316,E2 -15841.316} C_VEL
LIN {X 0,Y 305.668,Z 120.528,A -85,B 0,C 180,E1 -15845.277,E2 -15845.277} C_VEL
LIN {X 0,Y 305.747,Z 120.522,A -85,B 0,C 180,E1 -15847.927,E2 -15847.927} C_VEL
LIN {X 0,Y 305.6,Z 120.533,A -85,B 0,C 180,E1 -15851.945,E2 -15851.945} C_VEL
LIN {X 0,Y 305.639,Z 120.533,A -85,B 0,C 180,E1 -15855.035,E2 -15855.035} C_VEL
LIN {X 0,Y 305.577,Z 120.54,A -85,B 0,C 180,E1 -15859.445,E2 -15859.445} C_VEL
LIN {X 0,Y 305.492,Z 120.556,A -85,B 0,C 180,E1 -15863.041,E2 -15863.041} C_VEL
LIN {X 0,Y 305.548,Z 120.545,A -85,B 0,C 180,E1 -15866.227,E2 -15866.227} C_VEL
LIN {X 0,Y 305.496,Z 120.548,A -85,B 0,C 180,E1 -15869.05,E2 -15869.05} C_VEL
LIN {X 0,Y 305.444,Z 120.557,A -85,B 0,C 180,E1 -15871.952,E2 -15871.952} C_VEL
LIN {X 0,Y 305.463,Z 120.555,A -85,B 0,C 180,E1 -15875.113,E2 -15875.113} C_VEL
LIN {X 0,Y 305.441,Z 120.549,A -85,B 0,C 180,E1 -15878.526,E2 -15878.526} C_VEL
LIN {X 0,Y 305.455,Z 120.561,A -85,B 0,C 180,E1 -15882.586,E2 -15882.586} C_VEL
LIN {X 0,Y 305.474,Z 120.557,A -85,B 0,C 180,E1 -15887.41,E2 -15887.41} C_VEL
LIN {X 0,Y 305.5,Z 120.73,A -85,B 0,C 180,E1 -15890.274,E2 -15890.274} C_VEL
LIN {X 0,Y 308.219,Z 130.205,A -85,B 0,C 180,E1 -15893.64,E2 -15893.64} C_VEL
LIN {X 0,Y 309.961,Z 137.209,A -85,B 0,C 180,E1 -15895.962,E2 -15895.962} C_VEL
LIN {X 0,Y 319.363,Z 156.298,A -85,B 0,C 180,E1 -15897.711,E2 -15897.711} C_VEL
LIN {X 0,Y 324.316,Z 167.527,A -85,B 0,C 180,E1 -15898.608,E2 -15898.608} C_VEL
LIN {X 0,Y 327.696,Z 186.428,A -85,B 0,C 180,E1 -15899.487,E2 -15899.487} C_VEL
LIN {X 0,Y 324.68,Z 275.84,A -85,B 0,C 180,E1 -15901.474,E2 -15901.474} C_VEL
LIN {X 0,Y 323.483,Z 290.272,A -85,B 0,C 180,E1 -15902.021,E2 -15902.021} C_VEL
LIN {X 0,Y 321.862,Z 304.124,A -85,B 0,C 180,E1 -15902.795,E2 -15902.795} C_VEL
LIN {X 0,Y 319.98,Z 317.026,A -85,B 0,C 180,E1 -15903.767,E2 -15903.767} C_VEL
LIN {X 0,Y 317.917,Z 329.697,A -85,B 0,C 180,E1 -15905.007,E2 -15905.007} C_VEL
LIN {X 0,Y 315.529,Z 342.167,A -85,B 0,C 180,E1 -15906.538,E2 -15906.538} C_VEL
LIN {X 0,Y 313.127,Z 353.448,A -85,B 0,C 180,E1 -15908.264,E2 -15908.264} C_VEL
LIN {X 0,Y 310.83,Z 363.541,A -85,B 0,C 180,E1 -15910.174,E2 -15910.174} C_VEL
LIN {X 0,Y 308.858,Z 371.938,A -85,B 0,C 180,E1 -15912.11,E2 -15912.11} C_VEL
LIN {X 0,Y 307.086,Z 379.975,A -85,B 0,C 180,E1 -15914.4,E2 -15914.4} C_VEL
LIN {X 0,Y 305.706,Z 386.47,A -85,B 0,C 180,E1 -15916.709,E2 -15916.709} C_VEL
LIN {X 0,Y 304.552,Z 392.249,A -85,B 0,C 180,E1 -15919.361,E2 -15919.361} C_VEL
LIN {X 0,Y 303.912,Z 396.479,A -85,B 0,C 180,E1 -15922.024,E2 -15922.024} C_VEL
LIN {X 0,Y 303.617,Z 399.285,A -85,B 0,C 180,E1 -15924.687,E2 -15924.687} C_VEL
LIN {X 0,Y 303.587,Z 400.739,A -85,B 0,C 180,E1 -15927.346,E2 -15927.346} C_VEL
LIN {X 0,Y 303.562,Z 400.861,A -85,B 0,C 180,E1 -15930,E2 -15930} C_VEL
LIN {X 0,Y 303.593,Z 399.648,A -85,B 0,C 180,E1 -15932.653,E2 -15932.653} C_VEL
LIN {X 0,Y 303.596,Z 397.054,A -85,B 0,C 180,E1 -15935.313,E2 -15935.313} C_VEL
LIN {X 0,Y 303.833,Z 392.992,A -85,B 0,C 180,E1 -15937.977,E2 -15937.977} C_VEL
LIN {X 0,Y 304.359,Z 387.351,A -85,B 0,C 180,E1 -15940.645,E2 -15940.645} C_VEL
LIN {X 0,Y 305.242,Z 380.982,A -85,B 0,C 180,E1 -15942.972,E2 -15942.972} C_VEL
LIN {X 0,Y 306.207,Z 374.223,A -85,B 0,C 180,E1 -15944.98,E2 -15944.98} C_VEL
LIN {X 0,Y 307.338,Z 366.222,A -85,B 0,C 180,E1 -15946.951,E2 -15946.951} C_VEL
LIN {X 0,Y 308.938,Z 356.502,A -85,B 0,C 180,E1 -15948.915,E2 -15948.915} C_VEL
LIN {X 0,Y 310.726,Z 345.713,A -85,B 0,C 180,E1 -15950.696,E2 -15950.696} C_VEL
LIN {X 0,Y 312.602,Z 333.763,A -85,B 0,C 180,E1 -15952.296,E2 -15952.296} C_VEL
LIN {X 0,Y 314.144,Z 322.299,A -85,B 0,C 180,E1 -15953.54,E2 -15953.54} C_VEL
LIN {X 0,Y 315.725,Z 309.184,A -85,B 0,C 180,E1 -15954.669,E2 -15954.669} C_VEL
LIN {X 0,Y 317.096,Z 296.126,A -85,B 0,C 180,E1 -15955.518,E2 -15955.518} C_VEL
LIN {X 0,Y 318.19,Z 282.19,A -85,B 0,C 180,E1 -15956.171,E2 -15956.171} C_VEL
LIN {X 0,Y 318.853,Z 267.663,A -85,B 0,C 180,E1 -15956.597,E2 -15956.597} C_VEL
LIN {X 0,Y 320.987,Z 182.398,A -85,B 0,C 180,E1 -15958.489,E2 -15958.489} C_VEL
LIN {X 0,Y 316.586,Z 155.358,A -85,B 0,C 180,E1 -15959.548,E2 -15959.548} C_VEL
LIN {X 0,Y 309.403,Z 137.502,A -85,B 0,C 180,E1 -15960.715,E2 -15960.715} C_VEL
LIN {X 0,Y 307.167,Z 127.439,A -85,B 0,C 180,E1 -15963.677,E2 -15963.677} C_VEL
LIN {X 0,Y 305.492,Z 120.562,A -85,B 0,C 180,E1 -15965.817,E2 -15965.817} C_VEL
LIN {X 0,Y 305.466,Z 120.561,A -85,B 0,C 180,E1 -15968.533,E2 -15968.533} C_VEL
LIN {X 0,Y 305.462,Z 120.559,A -85,B 0,C 180,E1 -15972.587,E2 -15972.587} C_VEL
LIN {X 0,Y 305.492,Z 120.554,A -85,B 0,C 180,E1 -15976.357,E2 -15976.357} C_VEL
LIN {X 0,Y 305.482,Z 120.551,A -85,B 0,C 180,E1 -15979.896,E2 -15979.896} C_VEL
LIN {X 0,Y 305.498,Z 120.555,A -85,B 0,C 180,E1 -15983.627,E2 -15983.627} C_VEL
LIN {X 0,Y 305.463,Z 120.555,A -85,B 0,C 180,E1 -15986.483,E2 -15986.483} C_VEL
LIN {X 0,Y 305.494,Z 120.554,A -85,B 0,C 180,E1 -15990.95,E2 -15990.95} C_VEL
LIN {X 0,Y 305.571,Z 120.544,A -85,B 0,C 180,E1 -15994.088,E2 -15994.088} C_VEL
LIN {X 0,Y 305.5,Z 120.554,A -85,B 0,C 180,E1 -15998.403,E2 -15998.403} C_VEL
LIN {X 0,Y 305.589,Z 120.54,A -85,B 0,C 180,E1 -16001.218,E2 -16001.218} C_VEL
LIN {X 0,Y 305.648,Z 120.535,A -85,B 0,C 180,E1 -16005.349,E2 -16005.349} C_VEL
LIN {X 0,Y 305.637,Z 120.536,A -85,B 0,C 180,E1 -16009.4,E2 -16009.4} C_VEL
LIN {X 0,Y 305.795,Z 120.518,A -85,B 0,C 180,E1 -16012.074,E2 -16012.074} C_VEL
LIN {X 0,Y 305.685,Z 120.528,A -85,B 0,C 180,E1 -16014.724,E2 -16014.724} C_VEL
LIN {X 0,Y 305.954,Z 120.498,A -85,B 0,C 180,E1 -16018.684,E2 -16018.684} C_VEL
LIN {X 0,Y 305.954,Z 120.49,A -85,B 0,C 180,E1 -16021.316,E2 -16021.316} C_VEL
LIN {X 0,Y 305.675,Z 120.531,A -85,B 0,C 180,E1 -16025.277,E2 -16025.277} C_VEL
LIN {X 0,Y 305.764,Z 120.522,A -85,B 0,C 180,E1 -16027.927,E2 -16027.927} C_VEL
LIN {X 0,Y 305.603,Z 120.54,A -85,B 0,C 180,E1 -16031.945,E2 -16031.945} C_VEL
LIN {X 0,Y 305.637,Z 120.536,A -85,B 0,C 180,E1 -16035.035,E2 -16035.035} C_VEL
LIN {X 0,Y 305.576,Z 120.542,A -85,B 0,C 180,E1 -16039.445,E2 -16039.445} C_VEL
LIN {X 0,Y 305.491,Z 120.555,A -85,B 0,C 180,E1 -16043.042,E2 -16043.042} C_VEL
LIN {X 0,Y 305.531,Z 120.547,A -85,B 0,C 180,E1 -16046.221,E2 -16046.221} C_VEL
LIN {X 0,Y 305.488,Z 120.558,A -85,B 0,C 180,E1 -16049.048,E2 -16049.048} C_VEL
LIN {X 0,Y 305.442,Z 120.558,A -85,B 0,C 180,E1 -16051.953,E2 -16051.953} C_VEL
LIN {X 0,Y 305.462,Z 120.562,A -85,B 0,C 180,E1 -16055.114,E2 -16055.114} C_VEL
LIN {X 0,Y 305.44,Z 120.56,A -85,B 0,C 180,E1 -16058.527,E2 -16058.527} C_VEL
LIN {X 0,Y 305.46,Z 120.557,A -85,B 0,C 180,E1 -16062.587,E2 -16062.587} C_VEL
LIN {X 0,Y 305.443,Z 120.559,A -85,B 0,C 180,E1 -16066.348,E2 -16066.348} C_VEL
LIN {X 0,Y 305.459,Z 120.555,A -85,B 0,C 180,E1 -16069.893,E2 -16069.893} C_VEL
LIN {X 0,Y 305.481,Z 120.557,A -85,B 0,C 180,E1 -16073.632,E2 -16073.632} C_VEL
LIN {X 0,Y 305.466,Z 120.563,A -85,B 0,C 180,E1 -16076.484,E2 -16076.484} C_VEL
LIN {X 0,Y 305.432,Z 120.564,A -85,B 0,C 180,E1 -16079.588,E2 -16079.588} C_VEL
LIN {X 0,Y 305.477,Z 120.581,A -85,B 0,C 180,E1 -16083.433,E2 -16083.433} C_VEL
LIN {X 0,Y 306.742,Z 125.734,A -85,B 0,C 180,E1 -16085.119,E2 -16085.119} C_VEL
LIN {X 0,Y 316.045,Z 147.254,A -85,B 0,C 180,E1 -16086.574,E2 -16086.574} C_VEL
LIN {X 0,Y 321.117,Z 160.672,A -85,B 0,C 180,E1 -16087.366,E2 -16087.366} C_VEL
LIN {X 0,Y 321.567,Z 163.012,A -85,B 0,C 180,E1 -16087.463,E2 -16087.463} C_VEL
LIN {X 0,Y 318.85,Z 262.413,A -85,B 0,C 180,E1 -16089.687,E2 -16089.687} C_VEL
LIN {X 0,Y 318.15,Z 276.134,A -85,B 0,C 180,E1 -16090.23,E2 -16090.23} C_VEL
LIN {X 0,Y 317.055,Z 289.642,A -85,B 0,C 180,E1 -16091,E2 -16091} C_VEL
LIN {X 0,Y 315.626,Z 302.809,A -85,B 0,C 180,E1 -16092.004,E2 -16092.004} C_VEL
LIN {X 0,Y 314.213,Z 314.083,A -85,B 0,C 180,E1 -16093.096,E2 -16093.096} C_VEL
LIN {X 0,Y 312.523,Z 325.874,A -85,B 0,C 180,E1 -16094.512,E2 -16094.512} C_VEL
LIN {X 0,Y 311.001,Z 335.684,A -85,B 0,C 180,E1 -16095.941,E2 -16095.941} C_VEL
LIN {X 0,Y 309.252,Z 346.339,A -85,B 0,C 180,E1 -16097.832,E2 -16097.832} C_VEL
LIN {X 0,Y 307.75,Z 355.433,A -85,B 0,C 180,E1 -16099.806,E2 -16099.806} C_VEL
LIN {X 0,Y 306.5,Z 362.884,A -85,B 0,C 180,E1 -16101.761,E2 -16101.761} C_VEL
LIN {X 0,Y 305.385,Z 370.003,A -85,B 0,C 180,E1 -16104.056,E2 -16104.056} C_VEL
LIN {X 0,Y 304.589,Z 374.996,A -85,B 0,C 180,E1 -16106.031,E2 -16106.031} C_VEL
LIN {X 0,Y 304.002,Z 380.141,A -85,B 0,C 180,E1 -16108.676,E2 -16108.676} C_VEL
LIN {X 0,Y 303.648,Z 383.799,A -85,B 0,C 180,E1 -16111.326,E2 -16111.326} C_VEL
LIN {X 0,Y 303.623,Z 386.066,A -85,B 0,C 180,E1 -16113.982,E2 -16113.982} C_VEL
LIN {X 0,Y 303.594,Z 387.008,A -85,B 0,C 180,E1 -16116.647,E2 -16116.647} C_VEL
LIN {X 0,Y 303.549,Z 386.63,A -85,B 0,C 180,E1 -16119.327,E2 -16119.327} C_VEL
LIN {X 0,Y 303.894,Z 384.91,A -85,B 0,C 180,E1 -16122.013,E2 -16122.013} C_VEL
LIN {X 0,Y 304.549,Z 381.806,A -85,B 0,C 180,E1 -16124.705,E2 -16124.705} C_VEL
LIN {X 0,Y 305.461,Z 377.189,A -85,B 0,C 180,E1 -16127.404,E2 -16127.404} C_VEL
LIN {X 0,Y 306.525,Z 372.63,A -85,B 0,C 180,E1 -16129.418,E2 -16129.418} C_VEL
LIN {X 0,Y 308.077,Z 366.019,A -85,B 0,C 180,E1 -16131.759,E2 -16131.759} C_VEL
LIN {X 0,Y 310.091,Z 357.764,A -85,B 0,C 180,E1 -16134.077,E2 -16134.077} C_VEL
LIN {X 0,Y 312.027,Z 349.418,A -85,B 0,C 180,E1 -16135.982,E2 -16135.982} C_VEL
LIN {X 0,Y 313.956,Z 340.478,A -85,B 0,C 180,E1 -16137.678,E2 -16137.678} C_VEL
LIN {X 0,Y 316.143,Z 330.218,A -85,B 0,C 180,E1 -16139.28,E2 -16139.28} C_VEL
LIN {X 0,Y 318.309,Z 319.075,A -85,B 0,C 180,E1 -16140.703,E2 -16140.703} C_VEL
LIN {X 0,Y 320.375,Z 306.938,A -85,B 0,C 180,E1 -16141.953,E2 -16141.953} C_VEL
LIN {X 0,Y 322.284,Z 293.443,A -85,B 0,C 180,E1 -16143.037,E2 -16143.037} C_VEL
LIN {X 0,Y 323.732,Z 279.278,A -85,B 0,C 180,E1 -16143.894,E2 -16143.894} C_VEL
LIN {X 0,Y 324.886,Z 265.012,A -85,B 0,C 180,E1 -16144.477,E2 -16144.477} C_VEL
LIN {X 0,Y 325.709,Z 243.506,A -85,B 0,C 180,E1 -16145.006,E2 -16145.006} C_VEL
LIN {X 0,Y 328.172,Z 168.922,A -85,B 0,C 180,E1 -16146.636,E2 -16146.636} C_VEL
LIN {X 0,Y 323.013,Z 157.164,A -85,B 0,C 180,E1 -16147.548,E2 -16147.548} C_VEL
LIN {X 0,Y 320.11,Z 152.716,A -85,B 0,C 180,E1 -16148.02,E2 -16148.02} C_VEL
LIN {X 0,Y 307.959,Z 140.839,A -85,B 0,C 180,E1 -16149.938,E2 -16149.938} C_VEL
LIN {X 0,Y 305.295,Z 136.304,A -85,B 0,C 180,E1 -16150.441,E2 -16150.441} C_VEL
LIN {X 0,Y 301.368,Z 129.541,A -85,B 0,C 180,E1 -16151.209,E2 -16151.209} C_VEL
LIN {X 0,Y 299.701,Z 126.329,A -85,B 0,C 180,E1 -16151.565,E2 -16151.565} C_VEL
LIN {X 0,Y 298.381,Z 121.443,A -85,B 0,C 180,E1 -16153.553,E2 -16153.553} C_VEL
LIN {X 0,Y 298.371,Z 121.436,A -85,B 0,C 180,E1 -16156.915,E2 -16156.915} C_VEL
LIN {X 0,Y 298.352,Z 121.429,A -85,B 0,C 180,E1 -16161.019,E2 -16161.019} C_VEL
LIN {X 0,Y 298.405,Z 121.434,A -85,B 0,C 180,E1 -16163.928,E2 -16163.928} C_VEL
LIN {X 0,Y 298.394,Z 121.436,A -85,B 0,C 180,E1 -16167.199,E2 -16167.199} C_VEL
LIN {X 0,Y 298.403,Z 121.433,A -85,B 0,C 180,E1 -16170.625,E2 -16170.625} C_VEL
